	VAR robtarget OpenholeUD_2741 := [[495.65, -37.5, 189.61], [0.203301, 0.677251, 0.701328, -0.090218], [0,0,0,0], [9E9, 9E9, 9E9, 9E9, 9E9, 9E9]];
	VAR robtarget OpenholeUD_2742 := [[499.58, -37.5, 190.31], [0.21303, 0.674254, 0.699718, -0.101956], [0,0,0,0], [9E9, 9E9, 9E9, 9E9, 9E9, 9E9]];
	VAR robtarget OpenholeUD_2743 := [[503.52, -37.5, 191.01], [0.222381, 0.671228, 0.697958, -0.113376], [0,0,0,0], [9E9, 9E9, 9E9, 9E9, 9E9, 9E9]];
	VAR robtarget OpenholeUD_2744 := [[509.38, -37.5, 192.05], [0.183051, 0.683002, 0.683002, -0.183051], [0,0,0,0], [9E9, 9E9, 9E9, 9E9, 9E9, 9E9]];
	VAR robtarget OpenholeUD_2745 := [[513.38, -37.5, 192.04], [0.183051, 0.683002, 0.683002, -0.183051], [0,0,0,0], [9E9, 9E9, 9E9, 9E9, 9E9, 9E9]];
	VAR robtarget OpenholeUD_2746 := [[517.38, -37.5, 192.02], [0.183051, 0.683002, 0.683002, -0.183051], [0,0,0,0], [9E9, 9E9, 9E9, 9E9, 9E9, 9E9]];
	VAR robtarget OpenholeUD_2747 := [[521.38, -37.5, 192.01], [0.183051, 0.683002, 0.683002, -0.183051], [0,0,0,0], [9E9, 9E9, 9E9, 9E9, 9E9, 9E9]];
	VAR robtarget OpenholeUD_2748 := [[525.38, -37.5, 192], [0.183051, 0.683002, 0.683002, -0.183051], [0,0,0,0], [9E9, 9E9, 9E9, 9E9, 9E9, 9E9]];
	VAR robtarget OpenholeUD_2749 := [[529.38, -37.5, 191.99], [0.183051, 0.683002, 0.683002, -0.183051], [0,0,0,0], [9E9, 9E9, 9E9, 9E9, 9E9, 9E9]];
	VAR robtarget OpenholeUD_2750 := [[529.38, -37.5, 191.99], [0.183051, 0.683002, 0.683002, -0.183051], [0,0,0,0], [9E9, 9E9, 9E9, 9E9, 9E9, 9E9]];
	VAR robtarget OpenholeUD_2751 := [[529.38, -38.7, 192.68], [0.183051, 0.683002, 0.683002, -0.183051], [0,0,0,0], [9E9, 9E9, 9E9, 9E9, 9E9, 9E9]];
	VAR robtarget OpenholeUD_2752 := [[525.38, -38.7, 192.69], [0.183051, 0.683002, 0.683002, -0.183051], [0,0,0,0], [9E9, 9E9, 9E9, 9E9, 9E9, 9E9]];
	VAR robtarget OpenholeUD_2753 := [[521.38, -38.7, 192.71], [0.183051, 0.683002, 0.683002, -0.183051], [0,0,0,0], [9E9, 9E9, 9E9, 9E9, 9E9, 9E9]];
	VAR robtarget OpenholeUD_2754 := [[517.38, -38.7, 192.72], [0.183051, 0.683002, 0.683002, -0.183051], [0,0,0,0], [9E9, 9E9, 9E9, 9E9, 9E9, 9E9]];
	VAR robtarget OpenholeUD_2755 := [[513.38, -38.7, 192.73], [0.183051, 0.683002, 0.683002, -0.183051], [0,0,0,0], [9E9, 9E9, 9E9, 9E9, 9E9, 9E9]];
	VAR robtarget OpenholeUD_2756 := [[509.38, -38.7, 192.74], [0.183051, 0.683002, 0.683002, -0.183051], [0,0,0,0], [9E9, 9E9, 9E9, 9E9, 9E9, 9E9]];
	VAR robtarget OpenholeUD_2757 := [[505.45, -38.7, 192], [0.230133, 0.66861, 0.697627, -0.1154], [0,0,0,0], [9E9, 9E9, 9E9, 9E9, 9E9, 9E9]];
	VAR robtarget OpenholeUD_2758 := [[501.52, -38.7, 191.26], [0.221049, 0.671668, 0.699402, -0.104103], [0,0,0,0], [9E9, 9E9, 9E9, 9E9, 9E9, 9E9]];
	VAR robtarget OpenholeUD_2759 := [[497.59, -38.7, 190.51], [0.211589, 0.674707, 0.701032, -0.092485], [0,0,0,0], [9E9, 9E9, 9E9, 9E9, 9E9, 9E9]];
	VAR robtarget OpenholeUD_2760 := [[493.66, -38.7, 189.77], [0.20175, 0.677714, 0.702503, -0.080562], [0,0,0,0], [9E9, 9E9, 9E9, 9E9, 9E9, 9E9]];
	VAR robtarget OpenholeUD_2761 := [[489.73, -38.7, 189.02], [0.191532, 0.680673, 0.703796, -0.06835], [0,0,0,0], [9E9, 9E9, 9E9, 9E9, 9E9, 9E9]];
	VAR robtarget OpenholeUD_2762 := [[485.8, -38.7, 188.28], [0.180935, 0.683566, 0.704896, -0.055873], [0,0,0,0], [9E9, 9E9, 9E9, 9E9, 9E9, 9E9]];
	VAR robtarget OpenholeUD_2763 := [[481.87, -38.7, 187.54], [0.169961, 0.686377, 0.705788, -0.043162], [0,0,0,0], [9E9, 9E9, 9E9, 9E9, 9E9, 9E9]];
	VAR robtarget OpenholeUD_2764 := [[477.94, -38.7, 186.79], [0.158629, 0.689084, 0.70646, -0.030235], [0,0,0,0], [9E9, 9E9, 9E9, 9E9, 9E9, 9E9]];
	VAR robtarget OpenholeUD_2765 := [[474.01, -38.7, 186.05], [0.146953, 0.691668, 0.706899, -0.017125], [0,0,0,0], [9E9, 9E9, 9E9, 9E9, 9E9, 9E9]];
	VAR robtarget OpenholeUD_2766 := [[470.08, -38.7, 185.31], [0.134953, 0.694109, 0.707096, -0.003866], [0,0,0,0], [9E9, 9E9, 9E9, 9E9, 9E9, 9E9]];
	VAR robtarget OpenholeUD_2767 := [[466.15, -38.7, 184.56], [0.122651, 0.696388, 0.707043, 0.009503], [0,0,0,0], [9E9, 9E9, 9E9, 9E9, 9E9, 9E9]];
	VAR robtarget OpenholeUD_2768 := [[462.22, -38.7, 183.82], [0.110074, 0.698487, 0.706735, 0.02294], [0,0,0,0], [9E9, 9E9, 9E9, 9E9, 9E9, 9E9]];
	VAR robtarget OpenholeUD_2769 := [[458.29, -38.7, 183.07], [0.097255, 0.700387, 0.706169, 0.036403], [0,0,0,0], [9E9, 9E9, 9E9, 9E9, 9E9, 9E9]];
	VAR robtarget OpenholeUD_2770 := [[454.36, -38.7, 182.33], [0.084227, 0.702073, 0.705348, 0.049848], [0,0,0,0], [9E9, 9E9, 9E9, 9E9, 9E9, 9E9]];
	VAR robtarget OpenholeUD_2771 := [[450.43, -38.7, 181.59], [0.071029, 0.70353, 0.704274, 0.063232], [0,0,0,0], [9E9, 9E9, 9E9, 9E9, 9E9, 9E9]];
	VAR robtarget OpenholeUD_2772 := [[446.5, -38.7, 180.84], [0.05769, 0.70475, 0.702956, 0.0765], [0,0,0,0], [9E9, 9E9, 9E9, 9E9, 9E9, 9E9]];
	VAR robtarget OpenholeUD_2773 := [[442.57, -38.7, 180.1], [0.044257, 0.70572, 0.701405, 0.089614], [0,0,0,0], [9E9, 9E9, 9E9, 9E9, 9E9, 9E9]];
	VAR robtarget OpenholeUD_2774 := [[438.64, -38.7, 179.35], [0.030777, 0.706437, 0.699632, 0.102541], [0,0,0,0], [9E9, 9E9, 9E9, 9E9, 9E9, 9E9]];
	VAR robtarget OpenholeUD_2775 := [[434.71, -38.7, 178.61], [0.017296, 0.706895, 0.697653, 0.115242], [0,0,0,0], [9E9, 9E9, 9E9, 9E9, 9E9, 9E9]];
	VAR robtarget OpenholeUD_2776 := [[430.78, -38.7, 177.87], [0.003855, 0.707096, 0.695483, 0.127685], [0,0,0,0], [9E9, 9E9, 9E9, 9E9, 9E9, 9E9]];
	VAR robtarget OpenholeUD_2777 := [[426.85, -38.7, 177.12], [-0.009501, 0.707043, 0.693141, 0.139841], [0,0,0,0], [9E9, 9E9, 9E9, 9E9, 9E9, 9E9]];
	VAR robtarget OpenholeUD_2778 := [[422.92, -38.7, 176.38], [-0.022733, 0.706741, 0.690646, 0.151685], [0,0,0,0], [9E9, 9E9, 9E9, 9E9, 9E9, 9E9]];
	VAR robtarget OpenholeUD_2779 := [[418.99, -38.7, 175.64], [-0.035803, 0.7062, 0.688017, 0.163195], [0,0,0,0], [9E9, 9E9, 9E9, 9E9, 9E9, 9E9]];
	VAR robtarget OpenholeUD_2780 := [[415.06, -38.7, 174.89], [-0.048676, 0.705429, 0.685274, 0.174356], [0,0,0,0], [9E9, 9E9, 9E9, 9E9, 9E9, 9E9]];
	VAR robtarget OpenholeUD_2781 := [[411.13, -38.7, 174.15], [-0.061321, 0.704443, 0.682435, 0.185154], [0,0,0,0], [9E9, 9E9, 9E9, 9E9, 9E9, 9E9]];
	VAR robtarget OpenholeUD_2782 := [[407.2, -38.7, 173.4], [-0.073711, 0.703254, 0.67952, 0.195582], [0,0,0,0], [9E9, 9E9, 9E9, 9E9, 9E9, 9E9]];
	VAR robtarget OpenholeUD_2783 := [[403.27, -38.7, 172.66], [-0.085821, 0.701879, 0.676546, 0.205634], [0,0,0,0], [9E9, 9E9, 9E9, 9E9, 9E9, 9E9]];
	VAR robtarget OpenholeUD_2784 := [[399.34, -38.7, 171.92], [-0.097632, 0.700334, 0.67353, 0.215308], [0,0,0,0], [9E9, 9E9, 9E9, 9E9, 9E9, 9E9]];
	VAR robtarget OpenholeUD_2785 := [[395.41, -38.7, 171.17], [-0.109129, 0.698635, 0.670487, 0.224606], [0,0,0,0], [9E9, 9E9, 9E9, 9E9, 9E9, 9E9]];
	VAR robtarget OpenholeUD_2786 := [[389.31, -38.7, 170.02], [-0.126309, 0.695734, 0.665746, 0.238291], [0,0,0,0], [9E9, 9E9, 9E9, 9E9, 9E9, 9E9]];
	VAR robtarget OpenholeUD_2787 := [[385.31, -38.7, 170.03], [-0.183051, 0.683002, 0.683002, 0.183051], [0,0,0,0], [9E9, 9E9, 9E9, 9E9, 9E9, 9E9]];
	VAR robtarget OpenholeUD_2788 := [[381.31, -38.7, 170.05], [-0.183051, 0.683002, 0.683002, 0.183051], [0,0,0,0], [9E9, 9E9, 9E9, 9E9, 9E9, 9E9]];
	VAR robtarget OpenholeUD_2789 := [[377.31, -38.7, 170.06], [-0.183051, 0.683002, 0.683002, 0.183051], [0,0,0,0], [9E9, 9E9, 9E9, 9E9, 9E9, 9E9]];
	VAR robtarget OpenholeUD_2790 := [[373.31, -38.7, 170.07], [-0.183051, 0.683002, 0.683002, 0.183051], [0,0,0,0], [9E9, 9E9, 9E9, 9E9, 9E9, 9E9]];
	VAR robtarget OpenholeUD_2791 := [[369.31, -38.7, 170.08], [-0.183051, 0.683002, 0.683002, 0.183051], [0,0,0,0], [9E9, 9E9, 9E9, 9E9, 9E9, 9E9]];
	VAR robtarget OpenholeUD_2792 := [[369.31, -38.7, 170.08], [-0.183051, 0.683002, 0.683002, 0.183051], [0,0,0,0], [9E9, 9E9, 9E9, 9E9, 9E9, 9E9]];
	VAR robtarget OpenholeUD_2793 := [[369.31, -38.7, 170.2], [-0.183051, 0.683002, 0.683002, 0.183051], [0,0,0,0], [9E9, 9E9, 9E9, 9E9, 9E9, 9E9]];
	VAR robtarget OpenholeUD_2794 := [[373.31, -38.7, 170.19], [-0.183051, 0.683002, 0.683002, 0.183051], [0,0,0,0], [9E9, 9E9, 9E9, 9E9, 9E9, 9E9]];
	VAR robtarget OpenholeUD_2795 := [[377.31, -38.7, 170.18], [-0.183051, 0.683002, 0.683002, 0.183051], [0,0,0,0], [9E9, 9E9, 9E9, 9E9, 9E9, 9E9]];
	VAR robtarget OpenholeUD_2796 := [[381.31, -38.7, 170.17], [-0.183051, 0.683002, 0.683002, 0.183051], [0,0,0,0], [9E9, 9E9, 9E9, 9E9, 9E9, 9E9]];
	VAR robtarget OpenholeUD_2797 := [[385.31, -38.7, 170.15], [-0.183051, 0.683002, 0.683002, 0.183051], [0,0,0,0], [9E9, 9E9, 9E9, 9E9, 9E9, 9E9]];
	VAR robtarget OpenholeUD_2798 := [[389.31, -38.7, 170.14], [-0.126405, 0.695717, 0.665808, 0.238118], [0,0,0,0], [9E9, 9E9, 9E9, 9E9, 9E9, 9E9]];
	VAR robtarget OpenholeUD_2799 := [[393.24, -38.7, 170.88], [-0.115413, 0.697624, 0.668864, 0.229394], [0,0,0,0], [9E9, 9E9, 9E9, 9E9, 9E9, 9E9]];
	VAR robtarget OpenholeUD_2800 := [[397.17, -38.7, 171.63], [-0.104088, 0.699404, 0.671913, 0.220302], [0,0,0,0], [9E9, 9E9, 9E9, 9E9, 9E9, 9E9]];
	VAR robtarget OpenholeUD_2801 := [[401.1, -38.7, 172.37], [-0.092441, 0.701038, 0.674943, 0.210836], [0,0,0,0], [9E9, 9E9, 9E9, 9E9, 9E9, 9E9]];
	VAR robtarget OpenholeUD_2802 := [[405.03, -38.7, 173.12], [-0.080484, 0.702511, 0.677939, 0.200994], [0,0,0,0], [9E9, 9E9, 9E9, 9E9, 9E9, 9E9]];
	VAR robtarget OpenholeUD_2803 := [[408.96, -38.7, 173.86], [-0.068237, 0.703807, 0.680885, 0.190776], [0,0,0,0], [9E9, 9E9, 9E9, 9E9, 9E9, 9E9]];
	VAR robtarget OpenholeUD_2804 := [[412.89, -38.7, 174.6], [-0.055719, 0.704908, 0.683764, 0.180185], [0,0,0,0], [9E9, 9E9, 9E9, 9E9, 9E9, 9E9]];
	VAR robtarget OpenholeUD_2805 := [[416.82, -38.7, 175.35], [-0.042956, 0.705801, 0.686558, 0.169228], [0,0,0,0], [9E9, 9E9, 9E9, 9E9, 9E9, 9E9]];
	VAR robtarget OpenholeUD_2806 := [[420.75, -38.7, 176.09], [-0.029979, 0.706471, 0.689248, 0.157914], [0,0,0,0], [9E9, 9E9, 9E9, 9E9, 9E9, 9E9]];
	VAR robtarget OpenholeUD_2807 := [[424.68, -38.7, 176.83], [-0.016818, 0.706907, 0.691815, 0.146259], [0,0,0,0], [9E9, 9E9, 9E9, 9E9, 9E9, 9E9]];
	VAR robtarget OpenholeUD_2808 := [[428.61, -38.7, 177.58], [-0.003512, 0.707098, 0.69424, 0.13428], [0,0,0,0], [9E9, 9E9, 9E9, 9E9, 9E9, 9E9]];
	VAR robtarget OpenholeUD_2809 := [[432.54, -38.7, 178.32], [0.009901, 0.707037, 0.696502, 0.122002], [0,0,0,0], [9E9, 9E9, 9E9, 9E9, 9E9, 9E9]];
	VAR robtarget OpenholeUD_2810 := [[436.47, -38.7, 179.07], [0.02338, 0.70672, 0.698585, 0.109449], [0,0,0,0], [9E9, 9E9, 9E9, 9E9, 9E9, 9E9]];
	VAR robtarget OpenholeUD_2811 := [[440.4, -38.7, 179.81], [0.036881, 0.706144, 0.70047, 0.096654], [0,0,0,0], [9E9, 9E9, 9E9, 9E9, 9E9, 9E9]];
	VAR robtarget OpenholeUD_2812 := [[444.33, -38.7, 180.55], [0.050359, 0.705311, 0.702141, 0.083651], [0,0,0,0], [9E9, 9E9, 9E9, 9E9, 9E9, 9E9]];
	VAR robtarget OpenholeUD_2813 := [[448.26, -38.7, 181.3], [0.063771, 0.704225, 0.703586, 0.070478], [0,0,0,0], [9E9, 9E9, 9E9, 9E9, 9E9, 9E9]];
	VAR robtarget OpenholeUD_2814 := [[452.19, -38.7, 182.04], [0.077052, 0.702896, 0.704793, 0.057153], [0,0,0,0], [9E9, 9E9, 9E9, 9E9, 9E9, 9E9]];
	VAR robtarget OpenholeUD_2815 := [[456.12, -38.7, 182.78], [0.090178, 0.701333, 0.705753, 0.043736], [0,0,0,0], [9E9, 9E9, 9E9, 9E9, 9E9, 9E9]];
	VAR robtarget OpenholeUD_2816 := [[460.06, -38.7, 183.53], [0.103115, 0.699548, 0.706458, 0.030277], [0,0,0,0], [9E9, 9E9, 9E9, 9E9, 9E9, 9E9]];
	VAR robtarget OpenholeUD_2817 := [[463.99, -38.7, 184.27], [0.115828, 0.697556, 0.706907, 0.01682], [0,0,0,0], [9E9, 9E9, 9E9, 9E9, 9E9, 9E9]];
	VAR robtarget OpenholeUD_2818 := [[467.92, -38.7, 185.02], [0.128284, 0.695373, 0.707099, 0.003409], [0,0,0,0], [9E9, 9E9, 9E9, 9E9, 9E9, 9E9]];
	VAR robtarget OpenholeUD_2819 := [[471.85, -38.7, 185.76], [0.140451, 0.693018, 0.707037, -0.009914], [0,0,0,0], [9E9, 9E9, 9E9, 9E9, 9E9, 9E9]];
	VAR robtarget OpenholeUD_2820 := [[475.78, -38.7, 186.5], [0.152307, 0.690509, 0.706729, -0.02311], [0,0,0,0], [9E9, 9E9, 9E9, 9E9, 9E9, 9E9]];
	VAR robtarget OpenholeUD_2821 := [[479.71, -38.7, 187.25], [0.163828, 0.687867, 0.706183, -0.036142], [0,0,0,0], [9E9, 9E9, 9E9, 9E9, 9E9, 9E9]];
	VAR robtarget OpenholeUD_2822 := [[483.64, -38.7, 187.99], [0.174999, 0.68511, 0.705409, -0.048974], [0,0,0,0], [9E9, 9E9, 9E9, 9E9, 9E9, 9E9]];
	VAR robtarget OpenholeUD_2823 := [[487.57, -38.7, 188.73], [0.185806, 0.682258, 0.704421, -0.061577], [0,0,0,0], [9E9, 9E9, 9E9, 9E9, 9E9, 9E9]];
	VAR robtarget OpenholeUD_2824 := [[491.5, -38.7, 189.48], [0.196242, 0.67933, 0.703232, -0.073924], [0,0,0,0], [9E9, 9E9, 9E9, 9E9, 9E9, 9E9]];
	VAR robtarget OpenholeUD_2825 := [[495.43, -38.7, 190.22], [0.2063, 0.676343, 0.701859, -0.085991], [0,0,0,0], [9E9, 9E9, 9E9, 9E9, 9E9, 9E9]];
	VAR robtarget OpenholeUD_2826 := [[499.36, -38.7, 190.97], [0.21598, 0.673315, 0.700316, -0.09776], [0,0,0,0], [9E9, 9E9, 9E9, 9E9, 9E9, 9E9]];
	VAR robtarget OpenholeUD_2827 := [[503.29, -38.7, 191.71], [0.225282, 0.67026, 0.698621, -0.109216], [0,0,0,0], [9E9, 9E9, 9E9, 9E9, 9E9, 9E9]];
	VAR robtarget OpenholeUD_2828 := [[509.38, -38.7, 192.86], [0.183051, 0.683002, 0.683002, -0.183051], [0,0,0,0], [9E9, 9E9, 9E9, 9E9, 9E9, 9E9]];
	VAR robtarget OpenholeUD_2829 := [[513.38, -38.7, 192.85], [0.183051, 0.683002, 0.683002, -0.183051], [0,0,0,0], [9E9, 9E9, 9E9, 9E9, 9E9, 9E9]];
	VAR robtarget OpenholeUD_2830 := [[517.38, -38.7, 192.84], [0.183051, 0.683002, 0.683002, -0.183051], [0,0,0,0], [9E9, 9E9, 9E9, 9E9, 9E9, 9E9]];
	VAR robtarget OpenholeUD_2831 := [[521.38, -38.7, 192.83], [0.183051, 0.683002, 0.683002, -0.183051], [0,0,0,0], [9E9, 9E9, 9E9, 9E9, 9E9, 9E9]];
	VAR robtarget OpenholeUD_2832 := [[525.38, -38.7, 192.81], [0.183051, 0.683002, 0.683002, -0.183051], [0,0,0,0], [9E9, 9E9, 9E9, 9E9, 9E9, 9E9]];
	VAR robtarget OpenholeUD_2833 := [[529.38, -38.7, 192.8], [0.183051, 0.683002, 0.683002, -0.183051], [0,0,0,0], [9E9, 9E9, 9E9, 9E9, 9E9, 9E9]];
	VAR robtarget OpenholeUD_2834 := [[529.38, -38.7, 192.8], [0.183051, 0.683002, 0.683002, -0.183051], [0,0,0,0], [9E9, 9E9, 9E9, 9E9, 9E9, 9E9]];
	VAR robtarget OpenholeUD_2835 := [[529.38, -37.5, 192.11], [0.183051, 0.683002, 0.683002, -0.183051], [0,0,0,0], [9E9, 9E9, 9E9, 9E9, 9E9, 9E9]];
	VAR robtarget OpenholeUD_2836 := [[525.38, -37.5, 192.12], [0.183051, 0.683002, 0.683002, -0.183051], [0,0,0,0], [9E9, 9E9, 9E9, 9E9, 9E9, 9E9]];
	VAR robtarget OpenholeUD_2837 := [[521.38, -37.5, 192.13], [0.183051, 0.683002, 0.683002, -0.183051], [0,0,0,0], [9E9, 9E9, 9E9, 9E9, 9E9, 9E9]];
	VAR robtarget OpenholeUD_2838 := [[517.38, -37.5, 192.14], [0.183051, 0.683002, 0.683002, -0.183051], [0,0,0,0], [9E9, 9E9, 9E9, 9E9, 9E9, 9E9]];
	VAR robtarget OpenholeUD_2839 := [[513.38, -37.5, 192.16], [0.183051, 0.683002, 0.683002, -0.183051], [0,0,0,0], [9E9, 9E9, 9E9, 9E9, 9E9, 9E9]];
	VAR robtarget OpenholeUD_2840 := [[509.38, -37.5, 192.17], [0.183051, 0.683002, 0.683002, -0.183051], [0,0,0,0], [9E9, 9E9, 9E9, 9E9, 9E9, 9E9]];
	VAR robtarget OpenholeUD_2841 := [[505.44, -37.5, 191.47], [0.226975, 0.669688, 0.697068, -0.118728], [0,0,0,0], [9E9, 9E9, 9E9, 9E9, 9E9, 9E9]];
	VAR robtarget OpenholeUD_2842 := [[501.5, -37.5, 190.77], [0.217806, 0.672726, 0.698892, -0.107473], [0,0,0,0], [9E9, 9E9, 9E9, 9E9, 9E9, 9E9]];
	VAR robtarget OpenholeUD_2843 := [[497.57, -37.5, 190.07], [0.20826, 0.675742, 0.700574, -0.095895], [0,0,0,0], [9E9, 9E9, 9E9, 9E9, 9E9, 9E9]];
	VAR robtarget OpenholeUD_2844 := [[493.63, -37.5, 189.37], [0.198335, 0.678722, 0.702099, -0.084008], [0,0,0,0], [9E9, 9E9, 9E9, 9E9, 9E9, 9E9]];
	VAR robtarget OpenholeUD_2845 := [[489.69, -37.5, 188.67], [0.18803, 0.681649, 0.703449, -0.07183], [0,0,0,0], [9E9, 9E9, 9E9, 9E9, 9E9, 9E9]];
	VAR robtarget OpenholeUD_2846 := [[485.75, -37.5, 187.97], [0.177348, 0.684505, 0.704609, -0.05938], [0,0,0,0], [9E9, 9E9, 9E9, 9E9, 9E9, 9E9]];
	VAR robtarget OpenholeUD_2847 := [[481.81, -37.5, 187.27], [0.166298, 0.687274, 0.705564, -0.046684], [0,0,0,0], [9E9, 9E9, 9E9, 9E9, 9E9, 9E9]];
	VAR robtarget OpenholeUD_2848 := [[477.87, -37.5, 186.57], [0.154888, 0.689935, 0.7063, -0.03377], [0,0,0,0], [9E9, 9E9, 9E9, 9E9, 9E9, 9E9]];
	VAR robtarget OpenholeUD_2849 := [[473.94, -37.5, 185.87], [0.143135, 0.692468, 0.706805, -0.020671], [0,0,0,0], [9E9, 9E9, 9E9, 9E9, 9E9, 9E9]];
	VAR robtarget OpenholeUD_2850 := [[470, -37.5, 185.17], [0.131057, 0.694855, 0.707068, -0.007421], [0,0,0,0], [9E9, 9E9, 9E9, 9E9, 9E9, 9E9]];
	VAR robtarget OpenholeUD_2851 := [[466.06, -37.5, 184.47], [0.118677, 0.697077, 0.707082, 0.005939], [0,0,0,0], [9E9, 9E9, 9E9, 9E9, 9E9, 9E9]];
	VAR robtarget OpenholeUD_2852 := [[462.12, -37.5, 183.77], [0.106025, 0.699113, 0.706841, 0.01937], [0,0,0,0], [9E9, 9E9, 9E9, 9E9, 9E9, 9E9]];
	VAR robtarget OpenholeUD_2853 := [[458.18, -37.5, 183.07], [0.093131, 0.700947, 0.706344, 0.03283], [0,0,0,0], [9E9, 9E9, 9E9, 9E9, 9E9, 9E9]];
	VAR robtarget OpenholeUD_2854 := [[454.24, -37.5, 182.37], [0.08003, 0.702563, 0.705591, 0.046273], [0,0,0,0], [9E9, 9E9, 9E9, 9E9, 9E9, 9E9]];
	VAR robtarget OpenholeUD_2855 := [[450.31, -37.5, 181.67], [0.066762, 0.703948, 0.704586, 0.059657], [0,0,0,0], [9E9, 9E9, 9E9, 9E9, 9E9, 9E9]];
	VAR robtarget OpenholeUD_2856 := [[446.37, -37.5, 180.97], [0.053369, 0.70509, 0.703335, 0.072939], [0,0,0,0], [9E9, 9E9, 9E9, 9E9, 9E9, 9E9]];
	VAR robtarget OpenholeUD_2857 := [[442.43, -37.5, 180.27], [0.039892, 0.705981, 0.701848, 0.086077], [0,0,0,0], [9E9, 9E9, 9E9, 9E9, 9E9, 9E9]];
	VAR robtarget OpenholeUD_2858 := [[438.49, -37.5, 179.57], [0.026377, 0.706615, 0.700138, 0.099031], [0,0,0,0], [9E9, 9E9, 9E9, 9E9, 9E9, 9E9]];
	VAR robtarget OpenholeUD_2859 := [[434.55, -37.5, 178.87], [0.012867, 0.70699, 0.698218, 0.111765], [0,0,0,0], [9E9, 9E9, 9E9, 9E9, 9E9, 9E9]];
	VAR robtarget OpenholeUD_2860 := [[430.61, -37.5, 178.17], [-0.000592, 0.707107, 0.696106, 0.124246], [0,0,0,0], [9E9, 9E9, 9E9, 9E9, 9E9, 9E9]];
	VAR robtarget OpenholeUD_2861 := [[426.68, -37.5, 177.47], [-0.013959, 0.706969, 0.693818, 0.136443], [0,0,0,0], [9E9, 9E9, 9E9, 9E9, 9E9, 9E9]];
	VAR robtarget OpenholeUD_2862 := [[422.74, -37.5, 176.77], [-0.027193, 0.706584, 0.691374, 0.148332], [0,0,0,0], [9E9, 9E9, 9E9, 9E9, 9E9, 9E9]];
	VAR robtarget OpenholeUD_2863 := [[418.8, -37.5, 176.07], [-0.040257, 0.70596, 0.688792, 0.159891], [0,0,0,0], [9E9, 9E9, 9E9, 9E9, 9E9, 9E9]];
	VAR robtarget OpenholeUD_2864 := [[414.86, -37.5, 175.37], [-0.053115, 0.705109, 0.686093, 0.171103], [0,0,0,0], [9E9, 9E9, 9E9, 9E9, 9E9, 9E9]];
	VAR robtarget OpenholeUD_2865 := [[410.92, -37.5, 174.67], [-0.065738, 0.704044, 0.683295, 0.181955], [0,0,0,0], [9E9, 9E9, 9E9, 9E9, 9E9, 9E9]];
	VAR robtarget OpenholeUD_2866 := [[406.98, -37.5, 173.97], [-0.078098, 0.702781, 0.680417, 0.192438], [0,0,0,0], [9E9, 9E9, 9E9, 9E9, 9E9, 9E9]];
	VAR robtarget OpenholeUD_2867 := [[403.05, -37.5, 173.27], [-0.090172, 0.701334, 0.677477, 0.202547], [0,0,0,0], [9E9, 9E9, 9E9, 9E9, 9E9, 9E9]];
	VAR robtarget OpenholeUD_2868 := [[399.11, -37.5, 172.57], [-0.101941, 0.69972, 0.67449, 0.21228], [0,0,0,0], [9E9, 9E9, 9E9, 9E9, 9E9, 9E9]];
	VAR robtarget OpenholeUD_2869 := [[395.17, -37.5, 171.87], [-0.113391, 0.697956, 0.671473, 0.221638], [0,0,0,0], [9E9, 9E9, 9E9, 9E9, 9E9, 9E9]];
	VAR robtarget OpenholeUD_2870 := [[389.31, -37.5, 170.83], [-0.129802, 0.695091, 0.666961, 0.234869], [0,0,0,0], [9E9, 9E9, 9E9, 9E9, 9E9, 9E9]];
	VAR robtarget OpenholeUD_2871 := [[385.31, -37.5, 170.85], [-0.183051, 0.683002, 0.683002, 0.183051], [0,0,0,0], [9E9, 9E9, 9E9, 9E9, 9E9, 9E9]];
	VAR robtarget OpenholeUD_2872 := [[381.31, -37.5, 170.86], [-0.183051, 0.683002, 0.683002, 0.183051], [0,0,0,0], [9E9, 9E9, 9E9, 9E9, 9E9, 9E9]];
	VAR robtarget OpenholeUD_2873 := [[377.31, -37.5, 170.87], [-0.183051, 0.683002, 0.683002, 0.183051], [0,0,0,0], [9E9, 9E9, 9E9, 9E9, 9E9, 9E9]];
	VAR robtarget OpenholeUD_2874 := [[373.31, -37.5, 170.88], [-0.183051, 0.683002, 0.683002, 0.183051], [0,0,0,0], [9E9, 9E9, 9E9, 9E9, 9E9, 9E9]];
	VAR robtarget OpenholeUD_2875 := [[369.31, -37.5, 170.9], [-0.183051, 0.683002, 0.683002, 0.183051], [0,0,0,0], [9E9, 9E9, 9E9, 9E9, 9E9, 9E9]];
	VAR robtarget OpenholeUD_2876 := [[369.31, -37.5, 170.9], [-0.183051, 0.683002, 0.683002, 0.183051], [0,0,0,0], [9E9, 9E9, 9E9, 9E9, 9E9, 9E9]];
	VAR robtarget OpenholeUD_2877 := [[369.32, -36.3, 171.59], [-0.183051, 0.683002, 0.683002, 0.183051], [0,0,0,0], [9E9, 9E9, 9E9, 9E9, 9E9, 9E9]];
	VAR robtarget OpenholeUD_2878 := [[373.32, -36.3, 171.58], [-0.183051, 0.683002, 0.683002, 0.183051], [0,0,0,0], [9E9, 9E9, 9E9, 9E9, 9E9, 9E9]];
	VAR robtarget OpenholeUD_2879 := [[377.32, -36.3, 171.56], [-0.183051, 0.683002, 0.683002, 0.183051], [0,0,0,0], [9E9, 9E9, 9E9, 9E9, 9E9, 9E9]];
	VAR robtarget OpenholeUD_2880 := [[381.32, -36.3, 171.55], [-0.183051, 0.683002, 0.683002, 0.183051], [0,0,0,0], [9E9, 9E9, 9E9, 9E9, 9E9, 9E9]];
	VAR robtarget OpenholeUD_2881 := [[385.32, -36.3, 171.54], [-0.183051, 0.683002, 0.683002, 0.183051], [0,0,0,0], [9E9, 9E9, 9E9, 9E9, 9E9, 9E9]];
	VAR robtarget OpenholeUD_2882 := [[389.32, -36.3, 171.53], [-0.133206, 0.694447, 0.668101, 0.231606], [0,0,0,0], [9E9, 9E9, 9E9, 9E9, 9E9, 9E9]];
	VAR robtarget OpenholeUD_2883 := [[393.26, -36.3, 172.18], [-0.122294, 0.696451, 0.671117, 0.222715], [0,0,0,0], [9E9, 9E9, 9E9, 9E9, 9E9, 9E9]];
	VAR robtarget OpenholeUD_2884 := [[397.21, -36.3, 172.84], [-0.111044, 0.698333, 0.674119, 0.213456], [0,0,0,0], [9E9, 9E9, 9E9, 9E9, 9E9, 9E9]];
	VAR robtarget OpenholeUD_2885 := [[401.15, -36.3, 173.49], [-0.099464, 0.700076, 0.677094, 0.203822], [0,0,0,0], [9E9, 9E9, 9E9, 9E9, 9E9, 9E9]];
	VAR robtarget OpenholeUD_2886 := [[405.1, -36.3, 174.15], [-0.087567, 0.701664, 0.680027, 0.193813], [0,0,0,0], [9E9, 9E9, 9E9, 9E9, 9E9, 9E9]];
	VAR robtarget OpenholeUD_2887 := [[409.04, -36.3, 174.8], [-0.075371, 0.703078, 0.682901, 0.183428], [0,0,0,0], [9E9, 9E9, 9E9, 9E9, 9E9, 9E9]];
	VAR robtarget OpenholeUD_2888 := [[412.99, -36.3, 175.46], [-0.062895, 0.704304, 0.685699, 0.172674], [0,0,0,0], [9E9, 9E9, 9E9, 9E9, 9E9, 9E9]];
	VAR robtarget OpenholeUD_2889 := [[416.94, -36.3, 176.12], [-0.050166, 0.705325, 0.688404, 0.161556], [0,0,0,0], [9E9, 9E9, 9E9, 9E9, 9E9, 9E9]];
	VAR robtarget OpenholeUD_2890 := [[420.88, -36.3, 176.77], [-0.03721, 0.706127, 0.690995, 0.150088], [0,0,0,0], [9E9, 9E9, 9E9, 9E9, 9E9, 9E9]];
	VAR robtarget OpenholeUD_2891 := [[424.83, -36.3, 177.43], [-0.024062, 0.706697, 0.693453, 0.138284], [0,0,0,0], [9E9, 9E9, 9E9, 9E9, 9E9, 9E9]];
	VAR robtarget OpenholeUD_2892 := [[428.77, -36.3, 178.08], [-0.010756, 0.707025, 0.69576, 0.126164], [0,0,0,0], [9E9, 9E9, 9E9, 9E9, 9E9, 9E9]];
	VAR robtarget OpenholeUD_2893 := [[432.72, -36.3, 178.74], [0.002667, 0.707102, 0.697897, 0.113753], [0,0,0,0], [9E9, 9E9, 9E9, 9E9, 9E9, 9E9]];
	VAR robtarget OpenholeUD_2894 := [[436.67, -36.3, 179.39], [0.016167, 0.706922, 0.699845, 0.101079], [0,0,0,0], [9E9, 9E9, 9E9, 9E9, 9E9, 9E9]];
	VAR robtarget OpenholeUD_2895 := [[440.61, -36.3, 180.05], [0.029701, 0.706483, 0.701588, 0.088173], [0,0,0,0], [9E9, 9E9, 9E9, 9E9, 9E9, 9E9]];
	VAR robtarget OpenholeUD_2896 := [[444.56, -36.3, 180.71], [0.043222, 0.705785, 0.70311, 0.075072], [0,0,0,0], [9E9, 9E9, 9E9, 9E9, 9E9, 9E9]];
	VAR robtarget OpenholeUD_2897 := [[448.5, -36.3, 181.36], [0.056688, 0.704831, 0.7044, 0.061815], [0,0,0,0], [9E9, 9E9, 9E9, 9E9, 9E9, 9E9]];
	VAR robtarget OpenholeUD_2898 := [[452.45, -36.3, 182.02], [0.070054, 0.703628, 0.705446, 0.048442], [0,0,0,0], [9E9, 9E9, 9E9, 9E9, 9E9, 9E9]];
	VAR robtarget OpenholeUD_2899 := [[456.4, -36.3, 182.67], [0.083277, 0.702186, 0.70624, 0.034996], [0,0,0,0], [9E9, 9E9, 9E9, 9E9, 9E9, 9E9]];
	VAR robtarget OpenholeUD_2900 := [[460.34, -36.3, 183.33], [0.096317, 0.700516, 0.706779, 0.021521], [0,0,0,0], [9E9, 9E9, 9E9, 9E9, 9E9, 9E9]];
	VAR robtarget OpenholeUD_2901 := [[464.29, -36.3, 183.98], [0.109136, 0.698634, 0.707061, 0.008061], [0,0,0,0], [9E9, 9E9, 9E9, 9E9, 9E9, 9E9]];
	VAR robtarget OpenholeUD_2902 := [[468.23, -36.3, 184.64], [0.1217, 0.696555, 0.707087, -0.005341], [0,0,0,0], [9E9, 9E9, 9E9, 9E9, 9E9, 9E9]];
	VAR robtarget OpenholeUD_2903 := [[472.18, -36.3, 185.3], [0.133979, 0.694298, 0.706861, -0.018643], [0,0,0,0], [9E9, 9E9, 9E9, 9E9, 9E9, 9E9]];
	VAR robtarget OpenholeUD_2904 := [[476.12, -36.3, 185.95], [0.145948, 0.691881, 0.706391, -0.031805], [0,0,0,0], [9E9, 9E9, 9E9, 9E9, 9E9, 9E9]];
	VAR robtarget OpenholeUD_2905 := [[480.07, -36.3, 186.61], [0.157583, 0.689324, 0.705687, -0.044792], [0,0,0,0], [9E9, 9E9, 9E9, 9E9, 9E9, 9E9]];
	VAR robtarget OpenholeUD_2906 := [[484.02, -36.3, 187.26], [0.168868, 0.686647, 0.704759, -0.05757], [0,0,0,0], [9E9, 9E9, 9E9, 9E9, 9E9, 9E9]];
	VAR robtarget OpenholeUD_2907 := [[487.96, -36.3, 187.92], [0.17979, 0.683868, 0.703623, -0.070108], [0,0,0,0], [9E9, 9E9, 9E9, 9E9, 9E9, 9E9]];
	VAR robtarget OpenholeUD_2908 := [[491.91, -36.3, 188.57], [0.19034, 0.681007, 0.702292, -0.08238], [0,0,0,0], [9E9, 9E9, 9E9, 9E9, 9E9, 9E9]];
	VAR robtarget OpenholeUD_2909 := [[495.85, -36.3, 189.23], [0.200512, 0.678082, 0.700782, -0.094365], [0,0,0,0], [9E9, 9E9, 9E9, 9E9, 9E9, 9E9]];
	VAR robtarget OpenholeUD_2910 := [[499.8, -36.3, 189.89], [0.210305, 0.675109, 0.69911, -0.106044], [0,0,0,0], [9E9, 9E9, 9E9, 9E9, 9E9, 9E9]];
	VAR robtarget OpenholeUD_2911 := [[503.75, -36.3, 190.54], [0.219719, 0.672104, 0.697293, -0.117402], [0,0,0,0], [9E9, 9E9, 9E9, 9E9, 9E9, 9E9]];
	VAR robtarget OpenholeUD_2912 := [[509.38, -36.3, 191.48], [0.183051, 0.683002, 0.683002, -0.183051], [0,0,0,0], [9E9, 9E9, 9E9, 9E9, 9E9, 9E9]];
	VAR robtarget OpenholeUD_2913 := [[513.38, -36.3, 191.46], [0.183051, 0.683002, 0.683002, -0.183051], [0,0,0,0], [9E9, 9E9, 9E9, 9E9, 9E9, 9E9]];
	VAR robtarget OpenholeUD_2914 := [[517.38, -36.3, 191.45], [0.183051, 0.683002, 0.683002, -0.183051], [0,0,0,0], [9E9, 9E9, 9E9, 9E9, 9E9, 9E9]];
	VAR robtarget OpenholeUD_2915 := [[521.38, -36.3, 191.44], [0.183051, 0.683002, 0.683002, -0.183051], [0,0,0,0], [9E9, 9E9, 9E9, 9E9, 9E9, 9E9]];
	VAR robtarget OpenholeUD_2916 := [[525.38, -36.3, 191.43], [0.183051, 0.683002, 0.683002, -0.183051], [0,0,0,0], [9E9, 9E9, 9E9, 9E9, 9E9, 9E9]];
	VAR robtarget OpenholeUD_2917 := [[529.38, -36.3, 191.41], [0.183051, 0.683002, 0.683002, -0.183051], [0,0,0,0], [9E9, 9E9, 9E9, 9E9, 9E9, 9E9]];
	VAR robtarget OpenholeUD_2918 := [[529.38, -36.3, 191.41], [0.183051, 0.683002, 0.683002, -0.183051], [0,0,0,0], [9E9, 9E9, 9E9, 9E9, 9E9, 9E9]];
	VAR robtarget OpenholeUD_2919 := [[529.38, -35.1, 190.72], [0.183051, 0.683002, 0.683002, -0.183051], [0,0,0,0], [9E9, 9E9, 9E9, 9E9, 9E9, 9E9]];
	VAR robtarget OpenholeUD_2920 := [[525.38, -35.1, 190.73], [0.183051, 0.683002, 0.683002, -0.183051], [0,0,0,0], [9E9, 9E9, 9E9, 9E9, 9E9, 9E9]];
	VAR robtarget OpenholeUD_2921 := [[521.38, -35.1, 190.75], [0.183051, 0.683002, 0.683002, -0.183051], [0,0,0,0], [9E9, 9E9, 9E9, 9E9, 9E9, 9E9]];
	VAR robtarget OpenholeUD_2922 := [[517.38, -35.1, 190.76], [0.183051, 0.683002, 0.683002, -0.183051], [0,0,0,0], [9E9, 9E9, 9E9, 9E9, 9E9, 9E9]];
	VAR robtarget OpenholeUD_2923 := [[513.38, -35.1, 190.77], [0.183051, 0.683002, 0.683002, -0.183051], [0,0,0,0], [9E9, 9E9, 9E9, 9E9, 9E9, 9E9]];
	VAR robtarget OpenholeUD_2924 := [[509.38, -35.1, 190.78], [0.183051, 0.683002, 0.683002, -0.183051], [0,0,0,0], [9E9, 9E9, 9E9, 9E9, 9E9, 9E9]];
	VAR robtarget OpenholeUD_2925 := [[505.42, -35.1, 190.17], [0.220265, 0.671925, 0.695864, -0.125592], [0,0,0,0], [9E9, 9E9, 9E9, 9E9, 9E9, 9E9]];
	VAR robtarget OpenholeUD_2926 := [[501.47, -35.1, 189.56], [0.210928, 0.674914, 0.697789, -0.114414], [0,0,0,0], [9E9, 9E9, 9E9, 9E9, 9E9, 9E9]];
	VAR robtarget OpenholeUD_2927 := [[497.52, -35.1, 188.95], [0.201214, 0.677874, 0.699578, -0.102908], [0,0,0,0], [9E9, 9E9, 9E9, 9E9, 9E9, 9E9]];
	VAR robtarget OpenholeUD_2928 := [[493.56, -35.1, 188.34], [0.191121, 0.680788, 0.701216, -0.091085], [0,0,0,0], [9E9, 9E9, 9E9, 9E9, 9E9, 9E9]];
	VAR robtarget OpenholeUD_2929 := [[489.61, -35.1, 187.73], [0.180649, 0.683642, 0.702684, -0.078962], [0,0,0,0], [9E9, 9E9, 9E9, 9E9, 9E9, 9E9]];
	VAR robtarget OpenholeUD_2930 := [[485.66, -35.1, 187.12], [0.169804, 0.686416, 0.703967, -0.06656], [0,0,0,0], [9E9, 9E9, 9E9, 9E9, 9E9, 9E9]];
	VAR robtarget OpenholeUD_2931 := [[481.71, -35.1, 186.51], [0.158593, 0.689092, 0.705049, -0.053901], [0,0,0,0], [9E9, 9E9, 9E9, 9E9, 9E9, 9E9]];
	VAR robtarget OpenholeUD_2932 := [[477.75, -35.1, 185.89], [0.147029, 0.691652, 0.705916, -0.041015], [0,0,0,0], [9E9, 9E9, 9E9, 9E9, 9E9, 9E9]];
	VAR robtarget OpenholeUD_2933 := [[473.8, -35.1, 185.28], [0.135127, 0.694075, 0.706555, -0.027933], [0,0,0,0], [9E9, 9E9, 9E9, 9E9, 9E9, 9E9]];
	VAR robtarget OpenholeUD_2934 := [[469.85, -35.1, 184.67], [0.122908, 0.696343, 0.706954, -0.01469], [0,0,0,0], [9E9, 9E9, 9E9, 9E9, 9E9, 9E9]];
	VAR robtarget OpenholeUD_2935 := [[465.89, -35.1, 184.06], [0.110397, 0.698436, 0.707106, -0.001325], [0,0,0,0], [9E9, 9E9, 9E9, 9E9, 9E9, 9E9]];
	VAR robtarget OpenholeUD_2936 := [[461.94, -35.1, 183.45], [0.097624, 0.700335, 0.707003, 0.012122], [0,0,0,0], [9E9, 9E9, 9E9, 9E9, 9E9, 9E9]];
	VAR robtarget OpenholeUD_2937 := [[457.99, -35.1, 182.84], [0.084621, 0.702025, 0.706643, 0.025609], [0,0,0,0], [9E9, 9E9, 9E9, 9E9, 9E9, 9E9]];
	VAR robtarget OpenholeUD_2938 := [[454.03, -35.1, 182.23], [0.071424, 0.70349, 0.706025, 0.03909], [0,0,0,0], [9E9, 9E9, 9E9, 9E9, 9E9, 9E9]];
	VAR robtarget OpenholeUD_2939 := [[450.08, -35.1, 181.61], [0.058075, 0.704718, 0.705153, 0.052524], [0,0,0,0], [9E9, 9E9, 9E9, 9E9, 9E9, 9E9]];
	VAR robtarget OpenholeUD_2940 := [[446.13, -35.1, 181], [0.044615, 0.705698, 0.704033, 0.065864], [0,0,0,0], [9E9, 9E9, 9E9, 9E9, 9E9, 9E9]];
	VAR robtarget OpenholeUD_2941 := [[442.17, -35.1, 180.39], [0.031087, 0.706423, 0.702672, 0.079071], [0,0,0,0], [9E9, 9E9, 9E9, 9E9, 9E9, 9E9]];
	VAR robtarget OpenholeUD_2942 := [[438.22, -35.1, 179.78], [0.017537, 0.706889, 0.701083, 0.092103], [0,0,0,0], [9E9, 9E9, 9E9, 9E9, 9E9, 9E9]];
	VAR robtarget OpenholeUD_2943 := [[434.27, -35.1, 179.17], [0.00401, 0.707095, 0.699279, 0.104923], [0,0,0,0], [9E9, 9E9, 9E9, 9E9, 9E9, 9E9]];
	VAR robtarget OpenholeUD_2944 := [[430.32, -35.1, 178.56], [-0.009451, 0.707044, 0.697276, 0.117497], [0,0,0,0], [9E9, 9E9, 9E9, 9E9, 9E9, 9E9]];
	VAR robtarget OpenholeUD_2945 := [[426.36, -35.1, 177.95], [-0.022803, 0.706739, 0.695092, 0.129794], [0,0,0,0], [9E9, 9E9, 9E9, 9E9, 9E9, 9E9]];
	VAR robtarget OpenholeUD_2946 := [[422.41, -35.1, 177.34], [-0.036006, 0.706189, 0.692745, 0.141789], [0,0,0,0], [9E9, 9E9, 9E9, 9E9, 9E9, 9E9]];
	VAR robtarget OpenholeUD_2947 := [[418.46, -35.1, 176.72], [-0.049024, 0.705405, 0.690254, 0.153458], [0,0,0,0], [9E9, 9E9, 9E9, 9E9, 9E9, 9E9]];
	VAR robtarget OpenholeUD_2948 := [[414.5, -35.1, 176.11], [-0.061823, 0.704399, 0.687638, 0.164785], [0,0,0,0], [9E9, 9E9, 9E9, 9E9, 9E9, 9E9]];
	VAR robtarget OpenholeUD_2949 := [[410.55, -35.1, 175.5], [-0.074373, 0.703185, 0.684916, 0.175755], [0,0,0,0], [9E9, 9E9, 9E9, 9E9, 9E9, 9E9]];
	VAR robtarget OpenholeUD_2950 := [[406.6, -35.1, 174.89], [-0.086648, 0.701778, 0.682107, 0.186359], [0,0,0,0], [9E9, 9E9, 9E9, 9E9, 9E9, 9E9]];
	VAR robtarget OpenholeUD_2951 := [[402.64, -35.1, 174.28], [-0.098626, 0.700195, 0.679229, 0.19659], [0,0,0,0], [9E9, 9E9, 9E9, 9E9, 9E9, 9E9]];
	VAR robtarget OpenholeUD_2952 := [[398.69, -35.1, 173.67], [-0.110289, 0.698453, 0.676299, 0.206446], [0,0,0,0], [9E9, 9E9, 9E9, 9E9, 9E9, 9E9]];
	VAR robtarget OpenholeUD_2953 := [[394.74, -35.1, 173.06], [-0.121624, 0.696568, 0.673332, 0.215927], [0,0,0,0], [9E9, 9E9, 9E9, 9E9, 9E9, 9E9]];
	VAR robtarget OpenholeUD_2954 := [[389.32, -35.1, 172.22], [-0.136616, 0.693784, 0.669228, 0.228327], [0,0,0,0], [9E9, 9E9, 9E9, 9E9, 9E9, 9E9]];
	VAR robtarget OpenholeUD_2955 := [[385.32, -35.1, 172.23], [-0.183051, 0.683002, 0.683002, 0.183051], [0,0,0,0], [9E9, 9E9, 9E9, 9E9, 9E9, 9E9]];
	VAR robtarget OpenholeUD_2956 := [[381.32, -35.1, 172.24], [-0.183051, 0.683002, 0.683002, 0.183051], [0,0,0,0], [9E9, 9E9, 9E9, 9E9, 9E9, 9E9]];
	VAR robtarget OpenholeUD_2957 := [[377.32, -35.1, 172.26], [-0.183051, 0.683002, 0.683002, 0.183051], [0,0,0,0], [9E9, 9E9, 9E9, 9E9, 9E9, 9E9]];
	VAR robtarget OpenholeUD_2958 := [[373.32, -35.1, 172.27], [-0.183051, 0.683002, 0.683002, 0.183051], [0,0,0,0], [9E9, 9E9, 9E9, 9E9, 9E9, 9E9]];
	VAR robtarget OpenholeUD_2959 := [[369.32, -35.1, 172.28], [-0.183051, 0.683002, 0.683002, 0.183051], [0,0,0,0], [9E9, 9E9, 9E9, 9E9, 9E9, 9E9]];
	VAR robtarget OpenholeUD_2960 := [[369.32, -35.1, 172.28], [-0.183051, 0.683002, 0.683002, 0.183051], [0,0,0,0], [9E9, 9E9, 9E9, 9E9, 9E9, 9E9]];
	VAR robtarget OpenholeUD_2961 := [[369.32, -33.9, 172.97], [-0.183051, 0.683002, 0.683002, 0.183051], [0,0,0,0], [9E9, 9E9, 9E9, 9E9, 9E9, 9E9]];
	VAR robtarget OpenholeUD_2962 := [[373.32, -33.9, 172.96], [-0.183051, 0.683002, 0.683002, 0.183051], [0,0,0,0], [9E9, 9E9, 9E9, 9E9, 9E9, 9E9]];
	VAR robtarget OpenholeUD_2963 := [[377.32, -33.9, 172.95], [-0.183051, 0.683002, 0.683002, 0.183051], [0,0,0,0], [9E9, 9E9, 9E9, 9E9, 9E9, 9E9]];
	VAR robtarget OpenholeUD_2964 := [[381.32, -33.9, 172.94], [-0.183051, 0.683002, 0.683002, 0.183051], [0,0,0,0], [9E9, 9E9, 9E9, 9E9, 9E9, 9E9]];
	VAR robtarget OpenholeUD_2965 := [[385.32, -33.9, 172.92], [-0.183051, 0.683002, 0.683002, 0.183051], [0,0,0,0], [9E9, 9E9, 9E9, 9E9, 9E9, 9E9]];
	VAR robtarget OpenholeUD_2966 := [[389.32, -33.9, 172.91], [-0.140033, 0.693102, 0.670343, 0.225034], [0,0,0,0], [9E9, 9E9, 9E9, 9E9, 9E9, 9E9]];
	VAR robtarget OpenholeUD_2967 := [[393.28, -33.9, 173.48], [-0.12921, 0.695201, 0.673315, 0.21598], [0,0,0,0], [9E9, 9E9, 9E9, 9E9, 9E9, 9E9]];
	VAR robtarget OpenholeUD_2968 := [[397.24, -33.9, 174.05], [-0.118043, 0.697184, 0.676266, 0.206554], [0,0,0,0], [9E9, 9E9, 9E9, 9E9, 9E9, 9E9]];
	VAR robtarget OpenholeUD_2969 := [[401.2, -33.9, 174.61], [-0.10654, 0.699034, 0.679181, 0.196755], [0,0,0,0], [9E9, 9E9, 9E9, 9E9, 9E9, 9E9]];
	VAR robtarget OpenholeUD_2970 := [[405.16, -33.9, 175.18], [-0.094713, 0.700735, 0.682047, 0.186581], [0,0,0,0], [9E9, 9E9, 9E9, 9E9, 9E9, 9E9]];
	VAR robtarget OpenholeUD_2971 := [[409.12, -33.9, 175.74], [-0.082578, 0.702268, 0.684844, 0.176035], [0,0,0,0], [9E9, 9E9, 9E9, 9E9, 9E9, 9E9]];
	VAR robtarget OpenholeUD_2972 := [[413.08, -33.9, 176.31], [-0.070156, 0.703618, 0.687557, 0.165121], [0,0,0,0], [9E9, 9E9, 9E9, 9E9, 9E9, 9E9]];
	VAR robtarget OpenholeUD_2973 := [[417.04, -33.9, 176.88], [-0.057469, 0.704768, 0.690167, 0.153848], [0,0,0,0], [9E9, 9E9, 9E9, 9E9, 9E9, 9E9]];
	VAR robtarget OpenholeUD_2974 := [[421, -33.9, 177.44], [-0.044546, 0.705702, 0.692655, 0.14223], [0,0,0,0], [9E9, 9E9, 9E9, 9E9, 9E9, 9E9]];
	VAR robtarget OpenholeUD_2975 := [[424.96, -33.9, 178.01], [-0.031419, 0.706408, 0.695001, 0.130283], [0,0,0,0], [9E9, 9E9, 9E9, 9E9, 9E9, 9E9]];
	VAR robtarget OpenholeUD_2976 := [[428.92, -33.9, 178.58], [-0.018124, 0.706874, 0.697187, 0.118029], [0,0,0,0], [9E9, 9E9, 9E9, 9E9, 9E9, 9E9]];
	VAR robtarget OpenholeUD_2977 := [[432.88, -33.9, 179.14], [-0.004699, 0.707091, 0.699193, 0.105494], [0,0,0,0], [9E9, 9E9, 9E9, 9E9, 9E9, 9E9]];
	VAR robtarget OpenholeUD_2978 := [[436.84, -33.9, 179.71], [0.008814, 0.707052, 0.701003, 0.092705], [0,0,0,0], [9E9, 9E9, 9E9, 9E9, 9E9, 9E9]];
	VAR robtarget OpenholeUD_2979 := [[440.8, -33.9, 180.28], [0.022371, 0.706753, 0.702601, 0.079698], [0,0,0,0], [9E9, 9E9, 9E9, 9E9, 9E9, 9E9]];
	VAR robtarget OpenholeUD_2980 := [[444.75, -33.9, 180.84], [0.03593, 0.706193, 0.703972, 0.066509], [0,0,0,0], [9E9, 9E9, 9E9, 9E9, 9E9, 9E9]];
	VAR robtarget OpenholeUD_2981 := [[448.71, -33.9, 181.41], [0.049443, 0.705376, 0.705104, 0.053177], [0,0,0,0], [9E9, 9E9, 9E9, 9E9, 9E9, 9E9]];
	VAR robtarget OpenholeUD_2982 := [[452.67, -33.9, 181.98], [0.062867, 0.704307, 0.705989, 0.039745], [0,0,0,0], [9E9, 9E9, 9E9, 9E9, 9E9, 9E9]];
	VAR robtarget OpenholeUD_2983 := [[456.63, -33.9, 182.54], [0.076159, 0.702993, 0.706619, 0.026256], [0,0,0,0], [9E9, 9E9, 9E9, 9E9, 9E9, 9E9]];
	VAR robtarget OpenholeUD_2984 := [[460.59, -33.9, 183.11], [0.089277, 0.701448, 0.706992, 0.012754], [0,0,0,0], [9E9, 9E9, 9E9, 9E9, 9E9, 9E9]];
	VAR robtarget OpenholeUD_2985 := [[464.55, -33.9, 183.68], [0.102183, 0.699685, 0.707106, -0.000717], [0,0,0,0], [9E9, 9E9, 9E9, 9E9, 9E9, 9E9]];
	VAR robtarget OpenholeUD_2986 := [[468.51, -33.9, 184.24], [0.114842, 0.697719, 0.706966, -0.014114], [0,0,0,0], [9E9, 9E9, 9E9, 9E9, 9E9, 9E9]];
	VAR robtarget OpenholeUD_2987 := [[472.47, -33.9, 184.81], [0.127223, 0.695568, 0.706576, -0.027395], [0,0,0,0], [9E9, 9E9, 9E9, 9E9, 9E9, 9E9]];
	VAR robtarget OpenholeUD_2988 := [[476.43, -33.9, 185.38], [0.139299, 0.69325, 0.705945, -0.040522], [0,0,0,0], [9E9, 9E9, 9E9, 9E9, 9E9, 9E9]];
	VAR robtarget OpenholeUD_2989 := [[480.39, -33.9, 185.94], [0.151047, 0.690786, 0.705083, -0.053459], [0,0,0,0], [9E9, 9E9, 9E9, 9E9, 9E9, 9E9]];
	VAR robtarget OpenholeUD_2990 := [[484.35, -33.9, 186.51], [0.16245, 0.688193, 0.704004, -0.066172], [0,0,0,0], [9E9, 9E9, 9E9, 9E9, 9E9, 9E9]];
	VAR robtarget OpenholeUD_2991 := [[488.31, -33.9, 187.08], [0.173493, 0.685493, 0.702721, -0.078633], [0,0,0,0], [9E9, 9E9, 9E9, 9E9, 9E9, 9E9]];
	VAR robtarget OpenholeUD_2992 := [[492.27, -33.9, 187.64], [0.184165, 0.682703, 0.70125, -0.090818], [0,0,0,0], [9E9, 9E9, 9E9, 9E9, 9E9, 9E9]];
	VAR robtarget OpenholeUD_2993 := [[496.23, -33.9, 188.21], [0.194462, 0.679841, 0.699608, -0.102704], [0,0,0,0], [9E9, 9E9, 9E9, 9E9, 9E9, 9E9]];
	VAR robtarget OpenholeUD_2994 := [[500.19, -33.9, 188.78], [0.204381, 0.676926, 0.697812, -0.114275], [0,0,0,0], [9E9, 9E9, 9E9, 9E9, 9E9, 9E9]];
	VAR robtarget OpenholeUD_2995 := [[504.15, -33.9, 189.34], [0.213921, 0.673972, 0.695877, -0.125517], [0,0,0,0], [9E9, 9E9, 9E9, 9E9, 9E9, 9E9]];
	VAR robtarget OpenholeUD_2996 := [[509.37, -33.9, 190.09], [0.183051, 0.683002, 0.683002, -0.183051], [0,0,0,0], [9E9, 9E9, 9E9, 9E9, 9E9, 9E9]];
	VAR robtarget OpenholeUD_2997 := [[513.37, -33.9, 190.08], [0.183051, 0.683002, 0.683002, -0.183051], [0,0,0,0], [9E9, 9E9, 9E9, 9E9, 9E9, 9E9]];
	VAR robtarget OpenholeUD_2998 := [[517.37, -33.9, 190.07], [0.183051, 0.683002, 0.683002, -0.183051], [0,0,0,0], [9E9, 9E9, 9E9, 9E9, 9E9, 9E9]];
	VAR robtarget OpenholeUD_2999 := [[521.37, -33.9, 190.05], [0.183051, 0.683002, 0.683002, -0.183051], [0,0,0,0], [9E9, 9E9, 9E9, 9E9, 9E9, 9E9]];
	VAR robtarget OpenholeUD_3000 := [[525.37, -33.9, 190.04], [0.183051, 0.683002, 0.683002, -0.183051], [0,0,0,0], [9E9, 9E9, 9E9, 9E9, 9E9, 9E9]];
	VAR robtarget OpenholeUD_3001 := [[529.37, -33.9, 190.03], [0.183051, 0.683002, 0.683002, -0.183051], [0,0,0,0], [9E9, 9E9, 9E9, 9E9, 9E9, 9E9]];
	VAR robtarget OpenholeUD_3002 := [[529.37, -33.9, 190.03], [0.183051, 0.683002, 0.683002, -0.183051], [0,0,0,0], [9E9, 9E9, 9E9, 9E9, 9E9, 9E9]];
	VAR robtarget OpenholeUD_3003 := [[529.37, -32.7, 189.34], [0.183051, 0.683002, 0.683002, -0.183051], [0,0,0,0], [9E9, 9E9, 9E9, 9E9, 9E9, 9E9]];
	VAR robtarget OpenholeUD_3004 := [[525.37, -32.7, 189.35], [0.183051, 0.683002, 0.683002, -0.183051], [0,0,0,0], [9E9, 9E9, 9E9, 9E9, 9E9, 9E9]];
	VAR robtarget OpenholeUD_3005 := [[521.37, -32.7, 189.36], [0.183051, 0.683002, 0.683002, -0.183051], [0,0,0,0], [9E9, 9E9, 9E9, 9E9, 9E9, 9E9]];
	VAR robtarget OpenholeUD_3006 := [[517.37, -32.7, 189.37], [0.183051, 0.683002, 0.683002, -0.183051], [0,0,0,0], [9E9, 9E9, 9E9, 9E9, 9E9, 9E9]];
	VAR robtarget OpenholeUD_3007 := [[513.37, -32.7, 189.39], [0.183051, 0.683002, 0.683002, -0.183051], [0,0,0,0], [9E9, 9E9, 9E9, 9E9, 9E9, 9E9]];
	VAR robtarget OpenholeUD_3008 := [[509.37, -32.7, 189.4], [0.183051, 0.683002, 0.683002, -0.183051], [0,0,0,0], [9E9, 9E9, 9E9, 9E9, 9E9, 9E9]];
	VAR robtarget OpenholeUD_3009 := [[505.41, -32.7, 188.88], [0.213499, 0.674106, 0.694584, -0.132488], [0,0,0,0], [9E9, 9E9, 9E9, 9E9, 9E9, 9E9]];
	VAR robtarget OpenholeUD_3010 := [[501.44, -32.7, 188.35], [0.203996, 0.677042, 0.696608, -0.121398], [0,0,0,0], [9E9, 9E9, 9E9, 9E9, 9E9, 9E9]];
	VAR robtarget OpenholeUD_3011 := [[497.47, -32.7, 187.83], [0.194116, 0.67994, 0.698503, -0.109972], [0,0,0,0], [9E9, 9E9, 9E9, 9E9, 9E9, 9E9]];
	VAR robtarget OpenholeUD_3012 := [[493.51, -32.7, 187.31], [0.183858, 0.682786, 0.700252, -0.098223], [0,0,0,0], [9E9, 9E9, 9E9, 9E9, 9E9, 9E9]];
	VAR robtarget OpenholeUD_3013 := [[489.54, -32.7, 186.79], [0.173224, 0.685561, 0.701837, -0.086166], [0,0,0,0], [9E9, 9E9, 9E9, 9E9, 9E9, 9E9]];
	VAR robtarget OpenholeUD_3014 := [[485.58, -32.7, 186.27], [0.162219, 0.688248, 0.703243, -0.07382], [0,0,0,0], [9E9, 9E9, 9E9, 9E9, 9E9, 9E9]];
	VAR robtarget OpenholeUD_3015 := [[481.61, -32.7, 185.75], [0.150854, 0.690828, 0.704453, -0.061209], [0,0,0,0], [9E9, 9E9, 9E9, 9E9, 9E9, 9E9]];
	VAR robtarget OpenholeUD_3016 := [[477.65, -32.7, 185.22], [0.13914, 0.693282, 0.705451, -0.048361], [0,0,0,0], [9E9, 9E9, 9E9, 9E9, 9E9, 9E9]];
	VAR robtarget OpenholeUD_3017 := [[473.68, -32.7, 184.7], [0.127096, 0.695591, 0.706225, -0.035306], [0,0,0,0], [9E9, 9E9, 9E9, 9E9, 9E9, 9E9]];
	VAR robtarget OpenholeUD_3018 := [[469.71, -32.7, 184.18], [0.114744, 0.697735, 0.706762, -0.022079], [0,0,0,0], [9E9, 9E9, 9E9, 9E9, 9E9, 9E9]];
	VAR robtarget OpenholeUD_3019 := [[465.75, -32.7, 183.66], [0.10211, 0.699695, 0.707053, -0.008717], [0,0,0,0], [9E9, 9E9, 9E9, 9E9, 9E9, 9E9]];
	VAR robtarget OpenholeUD_3020 := [[461.78, -32.7, 183.14], [0.089224, 0.701455, 0.707091, 0.004737], [0,0,0,0], [9E9, 9E9, 9E9, 9E9, 9E9, 9E9]];
	VAR robtarget OpenholeUD_3021 := [[457.82, -32.7, 182.62], [0.076121, 0.702998, 0.706871, 0.018243], [0,0,0,0], [9E9, 9E9, 9E9, 9E9, 9E9, 9E9]];
	VAR robtarget OpenholeUD_3022 := [[453.85, -32.7, 182.09], [0.062839, 0.704309, 0.706393, 0.031755], [0,0,0,0], [9E9, 9E9, 9E9, 9E9, 9E9, 9E9]];
	VAR robtarget OpenholeUD_3023 := [[449.88, -32.7, 181.57], [0.049418, 0.705378, 0.705659, 0.045231], [0,0,0,0], [9E9, 9E9, 9E9, 9E9, 9E9, 9E9]];
	VAR robtarget OpenholeUD_3024 := [[445.92, -32.7, 181.05], [0.035902, 0.706195, 0.704672, 0.058625], [0,0,0,0], [9E9, 9E9, 9E9, 9E9, 9E9, 9E9]];
	VAR robtarget OpenholeUD_3025 := [[441.95, -32.7, 180.53], [0.022334, 0.706754, 0.703442, 0.071895], [0,0,0,0], [9E9, 9E9, 9E9, 9E9, 9E9, 9E9]];
	VAR robtarget OpenholeUD_3026 := [[437.99, -32.7, 180.01], [0.008761, 0.707053, 0.701979, 0.085001], [0,0,0,0], [9E9, 9E9, 9E9, 9E9, 9E9, 9E9]];
	VAR robtarget OpenholeUD_3027 := [[434.02, -32.7, 179.49], [-0.004773, 0.707091, 0.700296, 0.097904], [0,0,0,0], [9E9, 9E9, 9E9, 9E9, 9E9, 9E9]];
	VAR robtarget OpenholeUD_3028 := [[430.06, -32.7, 178.96], [-0.018225, 0.706872, 0.698408, 0.11057], [0,0,0,0], [9E9, 9E9, 9E9, 9E9, 9E9, 9E9]];
	VAR robtarget OpenholeUD_3029 := [[426.09, -32.7, 178.44], [-0.031552, 0.706402, 0.696333, 0.122966], [0,0,0,0], [9E9, 9E9, 9E9, 9E9, 9E9, 9E9]];
	VAR robtarget OpenholeUD_3030 := [[422.12, -32.7, 177.92], [-0.044715, 0.705692, 0.694087, 0.135066], [0,0,0,0], [9E9, 9E9, 9E9, 9E9, 9E9, 9E9]];
	VAR robtarget OpenholeUD_3031 := [[418.16, -32.7, 177.4], [-0.057678, 0.704751, 0.691691, 0.146846], [0,0,0,0], [9E9, 9E9, 9E9, 9E9, 9E9, 9E9]];
	VAR robtarget OpenholeUD_3032 := [[414.19, -32.7, 176.88], [-0.070407, 0.703593, 0.689162, 0.158289], [0,0,0,0], [9E9, 9E9, 9E9, 9E9, 9E9, 9E9]];
	VAR robtarget OpenholeUD_3033 := [[410.23, -32.7, 176.36], [-0.082875, 0.702233, 0.686521, 0.169378], [0,0,0,0], [9E9, 9E9, 9E9, 9E9, 9E9, 9E9]];
	VAR robtarget OpenholeUD_3034 := [[406.26, -32.7, 175.83], [-0.095057, 0.700688, 0.683785, 0.180104], [0,0,0,0], [9E9, 9E9, 9E9, 9E9, 9E9, 9E9]];
	VAR robtarget OpenholeUD_3035 := [[402.29, -32.7, 175.31], [-0.106932, 0.698975, 0.680973, 0.19046], [0,0,0,0], [9E9, 9E9, 9E9, 9E9, 9E9, 9E9]];
	VAR robtarget OpenholeUD_3036 := [[398.33, -32.7, 174.79], [-0.118483, 0.69711, 0.678102, 0.200443], [0,0,0,0], [9E9, 9E9, 9E9, 9E9, 9E9, 9E9]];
	VAR robtarget OpenholeUD_3037 := [[394.36, -32.7, 174.27], [-0.129698, 0.69511, 0.675188, 0.210051], [0,0,0,0], [9E9, 9E9, 9E9, 9E9, 9E9, 9E9]];
	VAR robtarget OpenholeUD_3038 := [[389.32, -32.7, 173.6], [-0.143454, 0.692402, 0.671444, 0.221728], [0,0,0,0], [9E9, 9E9, 9E9, 9E9, 9E9, 9E9]];
	VAR robtarget OpenholeUD_3039 := [[385.32, -32.7, 173.62], [-0.183051, 0.683002, 0.683002, 0.183051], [0,0,0,0], [9E9, 9E9, 9E9, 9E9, 9E9, 9E9]];
	VAR robtarget OpenholeUD_3040 := [[381.32, -32.7, 173.63], [-0.183051, 0.683002, 0.683002, 0.183051], [0,0,0,0], [9E9, 9E9, 9E9, 9E9, 9E9, 9E9]];
	VAR robtarget OpenholeUD_3041 := [[377.32, -32.7, 173.64], [-0.183051, 0.683002, 0.683002, 0.183051], [0,0,0,0], [9E9, 9E9, 9E9, 9E9, 9E9, 9E9]];
	VAR robtarget OpenholeUD_3042 := [[373.32, -32.7, 173.66], [-0.183051, 0.683002, 0.683002, 0.183051], [0,0,0,0], [9E9, 9E9, 9E9, 9E9, 9E9, 9E9]];
	VAR robtarget OpenholeUD_3043 := [[369.32, -32.7, 173.67], [-0.183051, 0.683002, 0.683002, 0.183051], [0,0,0,0], [9E9, 9E9, 9E9, 9E9, 9E9, 9E9]];
	VAR robtarget OpenholeUD_3044 := [[369.32, -32.7, 173.67], [-0.183051, 0.683002, 0.683002, 0.183051], [0,0,0,0], [9E9, 9E9, 9E9, 9E9, 9E9, 9E9]];
	VAR robtarget OpenholeUD_3045 := [[369.32, -31.5, 174.36], [-0.183051, 0.683002, 0.683002, 0.183051], [0,0,0,0], [9E9, 9E9, 9E9, 9E9, 9E9, 9E9]];
	VAR robtarget OpenholeUD_3046 := [[373.32, -31.5, 174.35], [-0.183051, 0.683002, 0.683002, 0.183051], [0,0,0,0], [9E9, 9E9, 9E9, 9E9, 9E9, 9E9]];
	VAR robtarget OpenholeUD_3047 := [[377.32, -31.5, 174.34], [-0.183051, 0.683002, 0.683002, 0.183051], [0,0,0,0], [9E9, 9E9, 9E9, 9E9, 9E9, 9E9]];
	VAR robtarget OpenholeUD_3048 := [[381.32, -31.5, 174.32], [-0.183051, 0.683002, 0.683002, 0.183051], [0,0,0,0], [9E9, 9E9, 9E9, 9E9, 9E9, 9E9]];
	VAR robtarget OpenholeUD_3049 := [[385.32, -31.5, 174.31], [-0.183051, 0.683002, 0.683002, 0.183051], [0,0,0,0], [9E9, 9E9, 9E9, 9E9, 9E9, 9E9]];
	VAR robtarget OpenholeUD_3050 := [[389.32, -31.5, 174.3], [-0.146879, 0.691684, 0.672531, 0.218409], [0,0,0,0], [9E9, 9E9, 9E9, 9E9, 9E9, 9E9]];
	VAR robtarget OpenholeUD_3051 := [[393.3, -31.5, 174.77], [-0.136154, 0.693875, 0.675454, 0.209192], [0,0,0,0], [9E9, 9E9, 9E9, 9E9, 9E9, 9E9]];
	VAR robtarget OpenholeUD_3052 := [[397.27, -31.5, 175.25], [-0.12508, 0.695956, 0.67835, 0.199604], [0,0,0,0], [9E9, 9E9, 9E9, 9E9, 9E9, 9E9]];
	VAR robtarget OpenholeUD_3053 := [[401.24, -31.5, 175.73], [-0.113663, 0.697912, 0.681202, 0.189642], [0,0,0,0], [9E9, 9E9, 9E9, 9E9, 9E9, 9E9]];
	VAR robtarget OpenholeUD_3054 := [[405.21, -31.5, 176.2], [-0.101916, 0.699724, 0.683995, 0.179307], [0,0,0,0], [9E9, 9E9, 9E9, 9E9, 9E9, 9E9]];
	VAR robtarget OpenholeUD_3055 := [[409.18, -31.5, 176.68], [-0.089853, 0.701375, 0.686712, 0.168602], [0,0,0,0], [9E9, 9E9, 9E9, 9E9, 9E9, 9E9]];
	VAR robtarget OpenholeUD_3056 := [[413.15, -31.5, 177.16], [-0.077493, 0.702848, 0.689335, 0.157534], [0,0,0,0], [9E9, 9E9, 9E9, 9E9, 9E9, 9E9]];
	VAR robtarget OpenholeUD_3057 := [[417.12, -31.5, 177.63], [-0.064859, 0.704126, 0.691846, 0.146112], [0,0,0,0], [9E9, 9E9, 9E9, 9E9, 9E9, 9E9]];
	VAR robtarget OpenholeUD_3058 := [[421.1, -31.5, 178.11], [-0.051979, 0.705194, 0.694226, 0.13435], [0,0,0,0], [9E9, 9E9, 9E9, 9E9, 9E9, 9E9]];
	VAR robtarget OpenholeUD_3059 := [[425.07, -31.5, 178.59], [-0.038884, 0.706037, 0.696456, 0.122268], [0,0,0,0], [9E9, 9E9, 9E9, 9E9, 9E9, 9E9]];
	VAR robtarget OpenholeUD_3060 := [[429.04, -31.5, 179.06], [-0.025609, 0.706643, 0.698516, 0.109887], [0,0,0,0], [9E9, 9E9, 9E9, 9E9, 9E9, 9E9]];
	VAR robtarget OpenholeUD_3061 := [[433.01, -31.5, 179.54], [-0.012193, 0.707002, 0.70039, 0.097234], [0,0,0,0], [9E9, 9E9, 9E9, 9E9, 9E9, 9E9]];
	VAR robtarget OpenholeUD_3062 := [[436.98, -31.5, 180.02], [0.001325, 0.707106, 0.702059, 0.084341], [0,0,0,0], [9E9, 9E9, 9E9, 9E9, 9E9, 9E9]];
	VAR robtarget OpenholeUD_3063 := [[440.95, -31.5, 180.49], [0.014899, 0.70695, 0.703509, 0.071242], [0,0,0,0], [9E9, 9E9, 9E9, 9E9, 9E9, 9E9]];
	VAR robtarget OpenholeUD_3064 := [[444.92, -31.5, 180.97], [0.028486, 0.706533, 0.704726, 0.057974], [0,0,0,0], [9E9, 9E9, 9E9, 9E9, 9E9, 9E9]];
	VAR robtarget OpenholeUD_3065 := [[448.9, -31.5, 181.45], [0.04204, 0.705856, 0.7057, 0.044578], [0,0,0,0], [9E9, 9E9, 9E9, 9E9, 9E9, 9E9]];
	VAR robtarget OpenholeUD_3066 := [[452.87, -31.5, 181.92], [0.055517, 0.704924, 0.706423, 0.031097], [0,0,0,0], [9E9, 9E9, 9E9, 9E9, 9E9, 9E9]];
	VAR robtarget OpenholeUD_3067 := [[456.84, -31.5, 182.4], [0.068872, 0.703745, 0.706888, 0.017575], [0,0,0,0], [9E9, 9E9, 9E9, 9E9, 9E9, 9E9]];
	VAR robtarget OpenholeUD_3068 := [[460.81, -31.5, 182.88], [0.082064, 0.702329, 0.707095, 0.004056], [0,0,0,0], [9E9, 9E9, 9E9, 9E9, 9E9, 9E9]];
	VAR robtarget OpenholeUD_3069 := [[464.78, -31.5, 183.35], [0.095053, 0.700689, 0.707044, -0.009416], [0,0,0,0], [9E9, 9E9, 9E9, 9E9, 9E9, 9E9]];
	VAR robtarget OpenholeUD_3070 := [[468.75, -31.5, 183.83], [0.107805, 0.698841, 0.706739, -0.022797], [0,0,0,0], [9E9, 9E9, 9E9, 9E9, 9E9, 9E9]];
	VAR robtarget OpenholeUD_3071 := [[472.73, -31.5, 184.31], [0.120286, 0.696801, 0.706187, -0.036048], [0,0,0,0], [9E9, 9E9, 9E9, 9E9, 9E9, 9E9]];
	VAR robtarget OpenholeUD_3072 := [[476.7, -31.5, 184.78], [0.132469, 0.694588, 0.705398, -0.049129], [0,0,0,0], [9E9, 9E9, 9E9, 9E9, 9E9, 9E9]];
	VAR robtarget OpenholeUD_3073 := [[480.67, -31.5, 185.26], [0.144331, 0.69222, 0.704383, -0.062006], [0,0,0,0], [9E9, 9E9, 9E9, 9E9, 9E9, 9E9]];
	VAR robtarget OpenholeUD_3074 := [[484.64, -31.5, 185.74], [0.155851, 0.689718, 0.703156, -0.074647], [0,0,0,0], [9E9, 9E9, 9E9, 9E9, 9E9, 9E9]];
	VAR robtarget OpenholeUD_3075 := [[488.61, -31.5, 186.21], [0.167016, 0.687099, 0.701731, -0.087024], [0,0,0,0], [9E9, 9E9, 9E9, 9E9, 9E9, 9E9]];
	VAR robtarget OpenholeUD_3076 := [[492.58, -31.5, 186.69], [0.177814, 0.684385, 0.700126, -0.099112], [0,0,0,0], [9E9, 9E9, 9E9, 9E9, 9E9, 9E9]];
	VAR robtarget OpenholeUD_3077 := [[496.55, -31.5, 187.17], [0.188238, 0.681591, 0.698357, -0.110893], [0,0,0,0], [9E9, 9E9, 9E9, 9E9, 9E9, 9E9]];
	VAR robtarget OpenholeUD_3078 := [[500.53, -31.5, 187.64], [0.198286, 0.678736, 0.696441, -0.12235], [0,0,0,0], [9E9, 9E9, 9E9, 9E9, 9E9, 9E9]];
	VAR robtarget OpenholeUD_3079 := [[504.5, -31.5, 188.12], [0.207955, 0.675836, 0.694396, -0.133472], [0,0,0,0], [9E9, 9E9, 9E9, 9E9, 9E9, 9E9]];
	VAR robtarget OpenholeUD_3080 := [[509.37, -31.5, 188.7], [0.183051, 0.683002, 0.683002, -0.183051], [0,0,0,0], [9E9, 9E9, 9E9, 9E9, 9E9, 9E9]];
	VAR robtarget OpenholeUD_3081 := [[513.37, -31.5, 188.69], [0.183051, 0.683002, 0.683002, -0.183051], [0,0,0,0], [9E9, 9E9, 9E9, 9E9, 9E9, 9E9]];
	VAR robtarget OpenholeUD_3082 := [[517.37, -31.5, 188.68], [0.183051, 0.683002, 0.683002, -0.183051], [0,0,0,0], [9E9, 9E9, 9E9, 9E9, 9E9, 9E9]];
	VAR robtarget OpenholeUD_3083 := [[521.37, -31.5, 188.67], [0.183051, 0.683002, 0.683002, -0.183051], [0,0,0,0], [9E9, 9E9, 9E9, 9E9, 9E9, 9E9]];
	VAR robtarget OpenholeUD_3084 := [[529.37, -31.5, 188.64], [0.183051, 0.683002, 0.683002, -0.183051], [0,0,0,0], [9E9, 9E9, 9E9, 9E9, 9E9, 9E9]];
	VAR robtarget OpenholeUD_3085 := [[529.37, -31.5, 188.64], [0.183051, 0.683002, 0.683002, -0.183051], [0,0,0,0], [9E9, 9E9, 9E9, 9E9, 9E9, 9E9]];
	VAR robtarget OpenholeUD_3086 := [[529.37, -30.3, 187.95], [0.183051, 0.683002, 0.683002, -0.183051], [0,0,0,0], [9E9, 9E9, 9E9, 9E9, 9E9, 9E9]];
	VAR robtarget OpenholeUD_3087 := [[525.37, -30.3, 187.96], [0.183051, 0.683002, 0.683002, -0.183051], [0,0,0,0], [9E9, 9E9, 9E9, 9E9, 9E9, 9E9]];
	VAR robtarget OpenholeUD_3088 := [[521.37, -30.3, 187.97], [0.183051, 0.683002, 0.683002, -0.183051], [0,0,0,0], [9E9, 9E9, 9E9, 9E9, 9E9, 9E9]];
	VAR robtarget OpenholeUD_3089 := [[517.37, -30.3, 187.99], [0.183051, 0.683002, 0.683002, -0.183051], [0,0,0,0], [9E9, 9E9, 9E9, 9E9, 9E9, 9E9]];
	VAR robtarget OpenholeUD_3090 := [[509.37, -30.3, 188.01], [0.183051, 0.683002, 0.683002, -0.183051], [0,0,0,0], [9E9, 9E9, 9E9, 9E9, 9E9, 9E9]];
	VAR robtarget OpenholeUD_3091 := [[505.39, -30.3, 187.58], [0.206682, 0.676227, 0.693228, -0.139411], [0,0,0,0], [9E9, 9E9, 9E9, 9E9, 9E9, 9E9]];
	VAR robtarget OpenholeUD_3092 := [[501.41, -30.3, 187.15], [0.197016, 0.679106, 0.695348, -0.128416], [0,0,0,0], [9E9, 9E9, 9E9, 9E9, 9E9, 9E9]];
	VAR robtarget OpenholeUD_3093 := [[497.44, -30.3, 186.72], [0.186974, 0.681939, 0.697347, -0.11708], [0,0,0,0], [9E9, 9E9, 9E9, 9E9, 9E9, 9E9]];
	VAR robtarget OpenholeUD_3094 := [[493.46, -30.3, 186.29], [0.176555, 0.68471, 0.699205, -0.105414], [0,0,0,0], [9E9, 9E9, 9E9, 9E9, 9E9, 9E9]];
	VAR robtarget OpenholeUD_3095 := [[489.48, -30.3, 185.86], [0.165763, 0.687403, 0.700907, -0.093433], [0,0,0,0], [9E9, 9E9, 9E9, 9E9, 9E9, 9E9]];
	VAR robtarget OpenholeUD_3096 := [[485.51, -30.3, 185.42], [0.154604, 0.689998, 0.702434, -0.081154], [0,0,0,0], [9E9, 9E9, 9E9, 9E9, 9E9, 9E9]];
	VAR robtarget OpenholeUD_3097 := [[481.53, -30.3, 184.99], [0.14309, 0.692478, 0.703771, -0.068601], [0,0,0,0], [9E9, 9E9, 9E9, 9E9, 9E9, 9E9]];
	VAR robtarget OpenholeUD_3098 := [[477.55, -30.3, 184.56], [0.131233, 0.694822, 0.704902, -0.0558], [0,0,0,0], [9E9, 9E9, 9E9, 9E9, 9E9, 9E9]];
	VAR robtarget OpenholeUD_3099 := [[473.58, -30.3, 184.13], [0.119055, 0.697012, 0.705811, -0.042782], [0,0,0,0], [9E9, 9E9, 9E9, 9E9, 9E9, 9E9]];
	VAR robtarget OpenholeUD_3100 := [[469.6, -30.3, 183.7], [0.106577, 0.699029, 0.706488, -0.02958], [0,0,0,0], [9E9, 9E9, 9E9, 9E9, 9E9, 9E9]];
	VAR robtarget OpenholeUD_3101 := [[465.62, -30.3, 183.27], [0.093828, 0.700854, 0.70692, -0.016232], [0,0,0,0], [9E9, 9E9, 9E9, 9E9, 9E9, 9E9]];
	VAR robtarget OpenholeUD_3102 := [[461.65, -30.3, 182.84], [0.080838, 0.702471, 0.707101, -0.002779], [0,0,0,0], [9E9, 9E9, 9E9, 9E9, 9E9, 9E9]];
	VAR robtarget OpenholeUD_3103 := [[457.67, -30.3, 182.4], [0.067645, 0.703864, 0.707025, 0.010737], [0,0,0,0], [9E9, 9E9, 9E9, 9E9, 9E9, 9E9]];
	VAR robtarget OpenholeUD_3104 := [[453.69, -30.3, 181.97], [0.054286, 0.70502, 0.70669, 0.024273], [0,0,0,0], [9E9, 9E9, 9E9, 9E9, 9E9, 9E9]];
	VAR robtarget OpenholeUD_3105 := [[449.72, -30.3, 181.54], [0.040804, 0.705928, 0.706097, 0.037784], [0,0,0,0], [9E9, 9E9, 9E9, 9E9, 9E9, 9E9]];
	VAR robtarget OpenholeUD_3106 := [[445.74, -30.3, 181.11], [0.027242, 0.706582, 0.705249, 0.051226], [0,0,0,0], [9E9, 9E9, 9E9, 9E9, 9E9, 9E9]];
	VAR robtarget OpenholeUD_3107 := [[441.76, -30.3, 180.68], [0.013646, 0.706975, 0.704154, 0.064555], [0,0,0,0], [9E9, 9E9, 9E9, 9E9, 9E9, 9E9]];
	VAR robtarget OpenholeUD_3108 := [[437.79, -30.3, 180.25], [0.000059, 0.707107, 0.702821, 0.07773], [0,0,0,0], [9E9, 9E9, 9E9, 9E9, 9E9, 9E9]];
	VAR robtarget OpenholeUD_3109 := [[433.81, -30.3, 179.82], [-0.013472, 0.706978, 0.701264, 0.090713], [0,0,0,0], [9E9, 9E9, 9E9, 9E9, 9E9, 9E9]];
	VAR robtarget OpenholeUD_3110 := [[429.83, -30.3, 179.38], [-0.026904, 0.706595, 0.699496, 0.103467], [0,0,0,0], [9E9, 9E9, 9E9, 9E9, 9E9, 9E9]];
	VAR robtarget OpenholeUD_3111 := [[425.86, -30.3, 178.95], [-0.040195, 0.705963, 0.697534, 0.11596], [0,0,0,0], [9E9, 9E9, 9E9, 9E9, 9E9, 9E9]];
	VAR robtarget OpenholeUD_3112 := [[421.88, -30.3, 178.52], [-0.053308, 0.705094, 0.695395, 0.128164], [0,0,0,0], [9E9, 9E9, 9E9, 9E9, 9E9, 9E9]];
	VAR robtarget OpenholeUD_3113 := [[417.9, -30.3, 178.09], [-0.066207, 0.704, 0.693098, 0.140056], [0,0,0,0], [9E9, 9E9, 9E9, 9E9, 9E9, 9E9]];
	VAR robtarget OpenholeUD_3114 := [[413.93, -30.3, 177.66], [-0.078859, 0.702696, 0.690661, 0.151614], [0,0,0,0], [9E9, 9E9, 9E9, 9E9, 9E9, 9E9]];
	VAR robtarget OpenholeUD_3115 := [[409.95, -30.3, 177.23], [-0.091238, 0.701196, 0.688105, 0.162825], [0,0,0,0], [9E9, 9E9, 9E9, 9E9, 9E9, 9E9]];
	VAR robtarget OpenholeUD_3116 := [[405.97, -30.3, 176.8], [-0.103319, 0.699518, 0.685447, 0.173675], [0,0,0,0], [9E9, 9E9, 9E9, 9E9, 9E9, 9E9]];
	VAR robtarget OpenholeUD_3117 := [[402, -30.3, 176.37], [-0.115084, 0.697679, 0.682705, 0.184158], [0,0,0,0], [9E9, 9E9, 9E9, 9E9, 9E9, 9E9]];
	VAR robtarget OpenholeUD_3118 := [[398.02, -30.3, 175.93], [-0.126517, 0.695696, 0.679897, 0.194269], [0,0,0,0], [9E9, 9E9, 9E9, 9E9, 9E9, 9E9]];
	VAR robtarget OpenholeUD_3119 := [[394.04, -30.3, 175.5], [-0.137607, 0.693588, 0.677039, 0.204006], [0,0,0,0], [9E9, 9E9, 9E9, 9E9, 9E9, 9E9]];
	VAR robtarget OpenholeUD_3120 := [[389.33, -30.3, 174.99], [-0.150308, 0.690947, 0.673603, 0.215078], [0,0,0,0], [9E9, 9E9, 9E9, 9E9, 9E9, 9E9]];
	VAR robtarget OpenholeUD_3121 := [[385.33, -30.3, 175], [-0.183051, 0.683002, 0.683002, 0.183051], [0,0,0,0], [9E9, 9E9, 9E9, 9E9, 9E9, 9E9]];
	VAR robtarget OpenholeUD_3122 := [[381.33, -30.3, 175.02], [-0.183051, 0.683002, 0.683002, 0.183051], [0,0,0,0], [9E9, 9E9, 9E9, 9E9, 9E9, 9E9]];
	VAR robtarget OpenholeUD_3123 := [[377.33, -30.3, 175.03], [-0.183051, 0.683002, 0.683002, 0.183051], [0,0,0,0], [9E9, 9E9, 9E9, 9E9, 9E9, 9E9]];
	VAR robtarget OpenholeUD_3124 := [[373.33, -30.3, 175.04], [-0.183051, 0.683002, 0.683002, 0.183051], [0,0,0,0], [9E9, 9E9, 9E9, 9E9, 9E9, 9E9]];
	VAR robtarget OpenholeUD_3125 := [[369.33, -30.3, 175.05], [-0.183051, 0.683002, 0.683002, 0.183051], [0,0,0,0], [9E9, 9E9, 9E9, 9E9, 9E9, 9E9]];
	VAR robtarget OpenholeUD_3126 := [[369.33, -30.3, 175.05], [-0.183051, 0.683002, 0.683002, 0.183051], [0,0,0,0], [9E9, 9E9, 9E9, 9E9, 9E9, 9E9]];
	VAR robtarget OpenholeUD_3127 := [[369.33, -29.1, 175.75], [-0.183051, 0.683002, 0.683002, 0.183051], [0,0,0,0], [9E9, 9E9, 9E9, 9E9, 9E9, 9E9]];
	VAR robtarget OpenholeUD_3128 := [[373.33, -29.1, 175.73], [-0.183051, 0.683002, 0.683002, 0.183051], [0,0,0,0], [9E9, 9E9, 9E9, 9E9, 9E9, 9E9]];
	VAR robtarget OpenholeUD_3129 := [[377.33, -29.1, 175.72], [-0.183051, 0.683002, 0.683002, 0.183051], [0,0,0,0], [9E9, 9E9, 9E9, 9E9, 9E9, 9E9]];
	VAR robtarget OpenholeUD_3130 := [[381.33, -29.1, 175.71], [-0.183051, 0.683002, 0.683002, 0.183051], [0,0,0,0], [9E9, 9E9, 9E9, 9E9, 9E9, 9E9]];
	VAR robtarget OpenholeUD_3131 := [[385.33, -29.1, 175.7], [-0.183051, 0.683002, 0.683002, 0.183051], [0,0,0,0], [9E9, 9E9, 9E9, 9E9, 9E9, 9E9]];
	VAR robtarget OpenholeUD_3132 := [[389.33, -29.1, 175.68], [-0.153739, 0.690191, 0.674661, 0.211736], [0,0,0,0], [9E9, 9E9, 9E9, 9E9, 9E9, 9E9]];
	VAR robtarget OpenholeUD_3133 := [[393.31, -29.1, 176.07], [-0.143121, 0.692471, 0.677533, 0.202358], [0,0,0,0], [9E9, 9E9, 9E9, 9E9, 9E9, 9E9]];
	VAR robtarget OpenholeUD_3134 := [[397.29, -29.1, 176.46], [-0.132148, 0.694649, 0.680368, 0.192611], [0,0,0,0], [9E9, 9E9, 9E9, 9E9, 9E9, 9E9]];
	VAR robtarget OpenholeUD_3135 := [[401.27, -29.1, 176.84], [-0.120827, 0.696707, 0.683152, 0.18249], [0,0,0,0], [9E9, 9E9, 9E9, 9E9, 9E9, 9E9]];
	VAR robtarget OpenholeUD_3136 := [[405.25, -29.1, 177.23], [-0.109169, 0.698629, 0.685869, 0.171999], [0,0,0,0], [9E9, 9E9, 9E9, 9E9, 9E9, 9E9]];
	VAR robtarget OpenholeUD_3137 := [[409.23, -29.1, 177.61], [-0.097187, 0.700396, 0.688501, 0.161141], [0,0,0,0], [9E9, 9E9, 9E9, 9E9, 9E9, 9E9]];
	VAR robtarget OpenholeUD_3138 := [[413.22, -29.1, 178], [-0.084899, 0.701992, 0.691031, 0.149923], [0,0,0,0], [9E9, 9E9, 9E9, 9E9, 9E9, 9E9]];
	VAR robtarget OpenholeUD_3139 := [[417.2, -29.1, 178.39], [-0.072329, 0.703398, 0.693439, 0.138357], [0,0,0,0], [9E9, 9E9, 9E9, 9E9, 9E9, 9E9]];
	VAR robtarget OpenholeUD_3140 := [[421.18, -29.1, 178.77], [-0.059502, 0.704599, 0.695707, 0.126459], [0,0,0,0], [9E9, 9E9, 9E9, 9E9, 9E9, 9E9]];
	VAR robtarget OpenholeUD_3141 := [[425.16, -29.1, 179.16], [-0.046449, 0.70558, 0.697816, 0.114248], [0,0,0,0], [9E9, 9E9, 9E9, 9E9, 9E9, 9E9]];
	VAR robtarget OpenholeUD_3142 := [[429.14, -29.1, 179.54], [-0.033204, 0.706327, 0.699748, 0.101748], [0,0,0,0], [9E9, 9E9, 9E9, 9E9, 9E9, 9E9]];
	VAR robtarget OpenholeUD_3143 := [[433.12, -29.1, 179.93], [-0.019805, 0.706829, 0.701485, 0.088987], [0,0,0,0], [9E9, 9E9, 9E9, 9E9, 9E9, 9E9]];
	VAR robtarget OpenholeUD_3144 := [[437.1, -29.1, 180.31], [-0.006293, 0.707079, 0.703011, 0.075998], [0,0,0,0], [9E9, 9E9, 9E9, 9E9, 9E9, 9E9]];
	VAR robtarget OpenholeUD_3145 := [[441.09, -29.1, 180.7], [0.007289, 0.707069, 0.704311, 0.062815], [0,0,0,0], [9E9, 9E9, 9E9, 9E9, 9E9, 9E9]];
	VAR robtarget OpenholeUD_3146 := [[445.07, -29.1, 181.09], [0.020897, 0.706798, 0.705374, 0.049478], [0,0,0,0], [9E9, 9E9, 9E9, 9E9, 9E9, 9E9]];
	VAR robtarget OpenholeUD_3147 := [[449.05, -29.1, 181.47], [0.034485, 0.706265, 0.706188, 0.036029], [0,0,0,0], [9E9, 9E9, 9E9, 9E9, 9E9, 9E9]];
	VAR robtarget OpenholeUD_3148 := [[453.03, -29.1, 181.86], [0.048007, 0.705475, 0.706748, 0.022509], [0,0,0,0], [9E9, 9E9, 9E9, 9E9, 9E9, 9E9]];
	VAR robtarget OpenholeUD_3149 := [[457.01, -29.1, 182.24], [0.06142, 0.704434, 0.70705, 0.008965], [0,0,0,0], [9E9, 9E9, 9E9, 9E9, 9E9, 9E9]];
	VAR robtarget OpenholeUD_3150 := [[460.99, -29.1, 182.63], [0.074682, 0.703152, 0.707092, -0.004561], [0,0,0,0], [9E9, 9E9, 9E9, 9E9, 9E9, 9E9]];
	VAR robtarget OpenholeUD_3151 := [[464.97, -29.1, 183.02], [0.087751, 0.701641, 0.706877, -0.018023], [0,0,0,0], [9E9, 9E9, 9E9, 9E9, 9E9, 9E9]];
	VAR robtarget OpenholeUD_3152 := [[468.96, -29.1, 183.4], [0.100592, 0.699915, 0.70641, -0.03138], [0,0,0,0], [9E9, 9E9, 9E9, 9E9, 9E9, 9E9]];
	VAR robtarget OpenholeUD_3153 := [[472.94, -29.1, 183.79], [0.113171, 0.697992, 0.705699, -0.04459], [0,0,0,0], [9E9, 9E9, 9E9, 9E9, 9E9, 9E9]];
	VAR robtarget OpenholeUD_3154 := [[476.92, -29.1, 184.17], [0.12546, 0.695888, 0.704755, -0.057617], [0,0,0,0], [9E9, 9E9, 9E9, 9E9, 9E9, 9E9]];
	VAR robtarget OpenholeUD_3155 := [[480.9, -29.1, 184.56], [0.137434, 0.693622, 0.703591, -0.070426], [0,0,0,0], [9E9, 9E9, 9E9, 9E9, 9E9, 9E9]];
	VAR robtarget OpenholeUD_3156 := [[484.88, -29.1, 184.95], [0.149073, 0.691214, 0.70222, -0.082986], [0,0,0,0], [9E9, 9E9, 9E9, 9E9, 9E9, 9E9]];
	VAR robtarget OpenholeUD_3157 := [[488.86, -29.1, 185.33], [0.16036, 0.688683, 0.700659, -0.095271], [0,0,0,0], [9E9, 9E9, 9E9, 9E9, 9E9, 9E9]];
	VAR robtarget OpenholeUD_3158 := [[492.84, -29.1, 185.72], [0.171285, 0.686048, 0.698925, -0.107257], [0,0,0,0], [9E9, 9E9, 9E9, 9E9, 9E9, 9E9]];
	VAR robtarget OpenholeUD_3159 := [[496.82, -29.1, 186.1], [0.181839, 0.683326, 0.697034, -0.118927], [0,0,0,0], [9E9, 9E9, 9E9, 9E9, 9E9, 9E9]];
	VAR robtarget OpenholeUD_3160 := [[500.81, -29.1, 186.49], [0.192017, 0.680536, 0.695004, -0.130266], [0,0,0,0], [9E9, 9E9, 9E9, 9E9, 9E9, 9E9]];
	VAR robtarget OpenholeUD_3161 := [[504.79, -29.1, 186.88], [0.201819, 0.677694, 0.692853, -0.141261], [0,0,0,0], [9E9, 9E9, 9E9, 9E9, 9E9, 9E9]];
	VAR robtarget OpenholeUD_3162 := [[509.37, -29.1, 187.32], [0.183051, 0.683002, 0.683002, -0.183051], [0,0,0,0], [9E9, 9E9, 9E9, 9E9, 9E9, 9E9]];
	VAR robtarget OpenholeUD_3163 := [[513.37, -29.1, 187.31], [0.183051, 0.683002, 0.683002, -0.183051], [0,0,0,0], [9E9, 9E9, 9E9, 9E9, 9E9, 9E9]];
	VAR robtarget OpenholeUD_3164 := [[517.37, -29.1, 187.29], [0.183051, 0.683002, 0.683002, -0.183051], [0,0,0,0], [9E9, 9E9, 9E9, 9E9, 9E9, 9E9]];
	VAR robtarget OpenholeUD_3165 := [[521.37, -29.1, 187.28], [0.183051, 0.683002, 0.683002, -0.183051], [0,0,0,0], [9E9, 9E9, 9E9, 9E9, 9E9, 9E9]];
	VAR robtarget OpenholeUD_3166 := [[529.37, -29.1, 187.26], [0.183051, 0.683002, 0.683002, -0.183051], [0,0,0,0], [9E9, 9E9, 9E9, 9E9, 9E9, 9E9]];
	VAR robtarget OpenholeUD_3167 := [[529.37, -29.1, 187.26], [0.183051, 0.683002, 0.683002, -0.183051], [0,0,0,0], [9E9, 9E9, 9E9, 9E9, 9E9, 9E9]];
	VAR robtarget OpenholeUD_3168 := [[529.36, -27.9, 186.56], [0.183051, 0.683002, 0.683002, -0.183051], [0,0,0,0], [9E9, 9E9, 9E9, 9E9, 9E9, 9E9]];
	VAR robtarget OpenholeUD_3169 := [[525.36, -27.9, 186.58], [0.183051, 0.683002, 0.683002, -0.183051], [0,0,0,0], [9E9, 9E9, 9E9, 9E9, 9E9, 9E9]];
	VAR robtarget OpenholeUD_3170 := [[521.36, -27.9, 186.59], [0.183051, 0.683002, 0.683002, -0.183051], [0,0,0,0], [9E9, 9E9, 9E9, 9E9, 9E9, 9E9]];
	VAR robtarget OpenholeUD_3171 := [[517.36, -27.9, 186.6], [0.183051, 0.683002, 0.683002, -0.183051], [0,0,0,0], [9E9, 9E9, 9E9, 9E9, 9E9, 9E9]];
	VAR robtarget OpenholeUD_3172 := [[509.36, -27.9, 186.63], [0.183051, 0.683002, 0.683002, -0.183051], [0,0,0,0], [9E9, 9E9, 9E9, 9E9, 9E9, 9E9]];
	VAR robtarget OpenholeUD_3173 := [[505.38, -27.9, 186.29], [0.19982, 0.678286, 0.691795, -0.146353], [0,0,0,0], [9E9, 9E9, 9E9, 9E9, 9E9, 9E9]];
	VAR robtarget OpenholeUD_3174 := [[501.39, -27.9, 185.95], [0.189995, 0.681103, 0.69401, -0.135463], [0,0,0,0], [9E9, 9E9, 9E9, 9E9, 9E9, 9E9]];
	VAR robtarget OpenholeUD_3175 := [[497.41, -27.9, 185.61], [0.179795, 0.683867, 0.696109, -0.124226], [0,0,0,0], [9E9, 9E9, 9E9, 9E9, 9E9, 9E9]];
	VAR robtarget OpenholeUD_3176 := [[493.42, -27.9, 185.26], [0.16922, 0.68656, 0.698076, -0.112652], [0,0,0,0], [9E9, 9E9, 9E9, 9E9, 9E9, 9E9]];
	VAR robtarget OpenholeUD_3177 := [[489.44, -27.9, 184.92], [0.158275, 0.689166, 0.699892, -0.100756], [0,0,0,0], [9E9, 9E9, 9E9, 9E9, 9E9, 9E9]];
	VAR robtarget OpenholeUD_3178 := [[485.45, -27.9, 184.58], [0.146967, 0.691665, 0.70154, -0.088554], [0,0,0,0], [9E9, 9E9, 9E9, 9E9, 9E9, 9E9]];
	VAR robtarget OpenholeUD_3179 := [[481.46, -27.9, 184.24], [0.13531, 0.69404, 0.703003, -0.076069], [0,0,0,0], [9E9, 9E9, 9E9, 9E9, 9E9, 9E9]];
	VAR robtarget OpenholeUD_3180 := [[477.48, -27.9, 183.9], [0.123318, 0.696271, 0.704266, -0.063325], [0,0,0,0], [9E9, 9E9, 9E9, 9E9, 9E9, 9E9]];
	VAR robtarget OpenholeUD_3181 := [[473.49, -27.9, 183.56], [0.111012, 0.698338, 0.705312, -0.050354], [0,0,0,0], [9E9, 9E9, 9E9, 9E9, 9E9, 9E9]];
	VAR robtarget OpenholeUD_3182 := [[469.51, -27.9, 183.22], [0.098417, 0.700224, 0.706128, -0.037187], [0,0,0,0], [9E9, 9E9, 9E9, 9E9, 9E9, 9E9]];
	VAR robtarget OpenholeUD_3183 := [[465.52, -27.9, 182.88], [0.085561, 0.701911, 0.706704, -0.023862], [0,0,0,0], [9E9, 9E9, 9E9, 9E9, 9E9, 9E9]];
	VAR robtarget OpenholeUD_3184 := [[461.54, -27.9, 182.54], [0.072478, 0.703383, 0.70703, -0.01042], [0,0,0,0], [9E9, 9E9, 9E9, 9E9, 9E9, 9E9]];
	VAR robtarget OpenholeUD_3185 := [[457.55, -27.9, 182.2], [0.059204, 0.704624, 0.7071, 0.003099], [0,0,0,0], [9E9, 9E9, 9E9, 9E9, 9E9, 9E9]];
	VAR robtarget OpenholeUD_3186 := [[453.57, -27.9, 181.86], [0.045779, 0.705623, 0.706911, 0.016651], [0,0,0,0], [9E9, 9E9, 9E9, 9E9, 9E9, 9E9]];
	VAR robtarget OpenholeUD_3187 := [[449.58, -27.9, 181.52], [0.032246, 0.706371, 0.706462, 0.03019], [0,0,0,0], [9E9, 9E9, 9E9, 9E9, 9E9, 9E9]];
	VAR robtarget OpenholeUD_3188 := [[445.6, -27.9, 181.18], [0.018649, 0.706861, 0.705757, 0.043672], [0,0,0,0], [9E9, 9E9, 9E9, 9E9, 9E9, 9E9]];
	VAR robtarget OpenholeUD_3189 := [[441.61, -27.9, 180.84], [0.005033, 0.707089, 0.704801, 0.057055], [0,0,0,0], [9E9, 9E9, 9E9, 9E9, 9E9, 9E9]];
	VAR robtarget OpenholeUD_3190 := [[437.62, -27.9, 180.5], [-0.008556, 0.707055, 0.703604, 0.070294], [0,0,0,0], [9E9, 9E9, 9E9, 9E9, 9E9, 9E9]];
	VAR robtarget OpenholeUD_3191 := [[433.64, -27.9, 180.16], [-0.022073, 0.706762, 0.702177, 0.083352], [0,0,0,0], [9E9, 9E9, 9E9, 9E9, 9E9, 9E9]];
	VAR robtarget OpenholeUD_3192 := [[429.65, -27.9, 179.82], [-0.035476, 0.706216, 0.700533, 0.096192], [0,0,0,0], [9E9, 9E9, 9E9, 9E9, 9E9, 9E9]];
	VAR robtarget OpenholeUD_3193 := [[425.67, -27.9, 179.48], [-0.048723, 0.705426, 0.698689, 0.10878], [0,0,0,0], [9E9, 9E9, 9E9, 9E9, 9E9, 9E9]];
	VAR robtarget OpenholeUD_3194 := [[421.68, -27.9, 179.14], [-0.061777, 0.704403, 0.696662, 0.121087], [0,0,0,0], [9E9, 9E9, 9E9, 9E9, 9E9, 9E9]];
	VAR robtarget OpenholeUD_3195 := [[417.7, -27.9, 178.8], [-0.074602, 0.70316, 0.694469, 0.133088], [0,0,0,0], [9E9, 9E9, 9E9, 9E9, 9E9, 9E9]];
	VAR robtarget OpenholeUD_3196 := [[413.71, -27.9, 178.46], [-0.08717, 0.701713, 0.69213, 0.144763], [0,0,0,0], [9E9, 9E9, 9E9, 9E9, 9E9, 9E9]];
	VAR robtarget OpenholeUD_3197 := [[409.73, -27.9, 178.12], [-0.099452, 0.700078, 0.689663, 0.156094], [0,0,0,0], [9E9, 9E9, 9E9, 9E9, 9E9, 9E9]];
	VAR robtarget OpenholeUD_3198 := [[405.74, -27.9, 177.78], [-0.111427, 0.698272, 0.687086, 0.16707], [0,0,0,0], [9E9, 9E9, 9E9, 9E9, 9E9, 9E9]];
	VAR robtarget OpenholeUD_3199 := [[401.75, -27.9, 177.44], [-0.123076, 0.696313, 0.684419, 0.177681], [0,0,0,0], [9E9, 9E9, 9E9, 9E9, 9E9, 9E9]];
	VAR robtarget OpenholeUD_3200 := [[397.77, -27.9, 177.1], [-0.134387, 0.694219, 0.681678, 0.187922], [0,0,0,0], [9E9, 9E9, 9E9, 9E9, 9E9, 9E9]];
	VAR robtarget OpenholeUD_3201 := [[393.78, -27.9, 176.76], [-0.145347, 0.692007, 0.67888, 0.197792], [0,0,0,0], [9E9, 9E9, 9E9, 9E9, 9E9, 9E9]];
	VAR robtarget OpenholeUD_3202 := [[389.33, -27.9, 176.38], [-0.157173, 0.689418, 0.675705, 0.208383], [0,0,0,0], [9E9, 9E9, 9E9, 9E9, 9E9, 9E9]];
	VAR robtarget OpenholeUD_3203 := [[385.33, -27.9, 176.39], [-0.183051, 0.683002, 0.683002, 0.183051], [0,0,0,0], [9E9, 9E9, 9E9, 9E9, 9E9, 9E9]];
	VAR robtarget OpenholeUD_3204 := [[381.33, -27.9, 176.4], [-0.183051, 0.683002, 0.683002, 0.183051], [0,0,0,0], [9E9, 9E9, 9E9, 9E9, 9E9, 9E9]];
	VAR robtarget OpenholeUD_3205 := [[377.33, -27.9, 176.41], [-0.183051, 0.683002, 0.683002, 0.183051], [0,0,0,0], [9E9, 9E9, 9E9, 9E9, 9E9, 9E9]];
	VAR robtarget OpenholeUD_3206 := [[373.33, -27.9, 176.43], [-0.183051, 0.683002, 0.683002, 0.183051], [0,0,0,0], [9E9, 9E9, 9E9, 9E9, 9E9, 9E9]];
	VAR robtarget OpenholeUD_3207 := [[369.33, -27.9, 176.44], [-0.183051, 0.683002, 0.683002, 0.183051], [0,0,0,0], [9E9, 9E9, 9E9, 9E9, 9E9, 9E9]];
	VAR robtarget OpenholeUD_3208 := [[369.33, -27.9, 176.44], [-0.183051, 0.683002, 0.683002, 0.183051], [0,0,0,0], [9E9, 9E9, 9E9, 9E9, 9E9, 9E9]];
	VAR robtarget OpenholeUD_3209 := [[369.33, -26.7, 177.13], [-0.183051, 0.683002, 0.683002, 0.183051], [0,0,0,0], [9E9, 9E9, 9E9, 9E9, 9E9, 9E9]];
	VAR robtarget OpenholeUD_3210 := [[373.33, -26.7, 177.12], [-0.183051, 0.683002, 0.683002, 0.183051], [0,0,0,0], [9E9, 9E9, 9E9, 9E9, 9E9, 9E9]];
	VAR robtarget OpenholeUD_3211 := [[377.33, -26.7, 177.11], [-0.183051, 0.683002, 0.683002, 0.183051], [0,0,0,0], [9E9, 9E9, 9E9, 9E9, 9E9, 9E9]];
	VAR robtarget OpenholeUD_3212 := [[381.33, -26.7, 177.1], [-0.183051, 0.683002, 0.683002, 0.183051], [0,0,0,0], [9E9, 9E9, 9E9, 9E9, 9E9, 9E9]];
	VAR robtarget OpenholeUD_3213 := [[385.33, -26.7, 177.08], [-0.183051, 0.683002, 0.683002, 0.183051], [0,0,0,0], [9E9, 9E9, 9E9, 9E9, 9E9, 9E9]];
	VAR robtarget OpenholeUD_3214 := [[389.33, -26.7, 177.07], [-0.160608, 0.688626, 0.676733, 0.205019], [0,0,0,0], [9E9, 9E9, 9E9, 9E9, 9E9, 9E9]];
	VAR robtarget OpenholeUD_3215 := [[393.32, -26.7, 177.36], [-0.150104, 0.690991, 0.679548, 0.195485], [0,0,0,0], [9E9, 9E9, 9E9, 9E9, 9E9, 9E9]];
	VAR robtarget OpenholeUD_3216 := [[397.31, -26.7, 177.66], [-0.13924, 0.693262, 0.682319, 0.185582], [0,0,0,0], [9E9, 9E9, 9E9, 9E9, 9E9, 9E9]];
	VAR robtarget OpenholeUD_3217 := [[401.3, -26.7, 177.95], [-0.128024, 0.695421, 0.685031, 0.175307], [0,0,0,0], [9E9, 9E9, 9E9, 9E9, 9E9, 9E9]];
	VAR robtarget OpenholeUD_3218 := [[405.29, -26.7, 178.25], [-0.116464, 0.69745, 0.687667, 0.164664], [0,0,0,0], [9E9, 9E9, 9E9, 9E9, 9E9, 9E9]];
	VAR robtarget OpenholeUD_3219 := [[409.28, -26.7, 178.54], [-0.104573, 0.699331, 0.69021, 0.153657], [0,0,0,0], [9E9, 9E9, 9E9, 9E9, 9E9, 9E9]];
	VAR robtarget OpenholeUD_3220 := [[413.27, -26.7, 178.84], [-0.092368, 0.701048, 0.692641, 0.142297], [0,0,0,0], [9E9, 9E9, 9E9, 9E9, 9E9, 9E9]];
	VAR robtarget OpenholeUD_3221 := [[417.26, -26.7, 179.13], [-0.079871, 0.702581, 0.694943, 0.130594], [0,0,0,0], [9E9, 9E9, 9E9, 9E9, 9E9, 9E9]];
	VAR robtarget OpenholeUD_3222 := [[421.25, -26.7, 179.43], [-0.067107, 0.703915, 0.697095, 0.118566], [0,0,0,0], [9E9, 9E9, 9E9, 9E9, 9E9, 9E9]];
	VAR robtarget OpenholeUD_3223 := [[425.23, -26.7, 179.72], [-0.054105, 0.705034, 0.699081, 0.106234], [0,0,0,0], [9E9, 9E9, 9E9, 9E9, 9E9, 9E9]];
	VAR robtarget OpenholeUD_3224 := [[429.22, -26.7, 180.02], [-0.0409, 0.705923, 0.700881, 0.093623], [0,0,0,0], [9E9, 9E9, 9E9, 9E9, 9E9, 9E9]];
	VAR robtarget OpenholeUD_3225 := [[433.21, -26.7, 180.31], [-0.027529, 0.706571, 0.702479, 0.080763], [0,0,0,0], [9E9, 9E9, 9E9, 9E9, 9E9, 9E9]];
	VAR robtarget OpenholeUD_3226 := [[437.2, -26.7, 180.6], [-0.014031, 0.706968, 0.70386, 0.067687], [0,0,0,0], [9E9, 9E9, 9E9, 9E9, 9E9, 9E9]];
	VAR robtarget OpenholeUD_3227 := [[441.19, -26.7, 180.9], [-0.00045, 0.707107, 0.705009, 0.054431], [0,0,0,0], [9E9, 9E9, 9E9, 9E9, 9E9, 9E9]];
	VAR robtarget OpenholeUD_3228 := [[445.18, -26.7, 181.19], [0.01317, 0.706984, 0.705915, 0.041035], [0,0,0,0], [9E9, 9E9, 9E9, 9E9, 9E9, 9E9]];
	VAR robtarget OpenholeUD_3229 := [[449.17, -26.7, 181.49], [0.026784, 0.706599, 0.70657, 0.027541], [0,0,0,0], [9E9, 9E9, 9E9, 9E9, 9E9, 9E9]];
	VAR robtarget OpenholeUD_3230 := [[453.16, -26.7, 181.78], [0.040345, 0.705955, 0.706968, 0.013993], [0,0,0,0], [9E9, 9E9, 9E9, 9E9, 9E9, 9E9]];
	VAR robtarget OpenholeUD_3231 := [[457.15, -26.7, 182.08], [0.05381, 0.705056, 0.707107, 0.000436], [0,0,0,0], [9E9, 9E9, 9E9, 9E9, 9E9, 9E9]];
	VAR robtarget OpenholeUD_3232 := [[461.14, -26.7, 182.37], [0.067135, 0.703913, 0.706986, -0.013086], [0,0,0,0], [9E9, 9E9, 9E9, 9E9, 9E9, 9E9]];
	VAR robtarget OpenholeUD_3233 := [[465.13, -26.7, 182.67], [0.08028, 0.702535, 0.706609, -0.026529], [0,0,0,0], [9E9, 9E9, 9E9, 9E9, 9E9, 9E9]];
	VAR robtarget OpenholeUD_3234 := [[469.12, -26.7, 182.96], [0.093207, 0.700937, 0.705983, -0.039852], [0,0,0,0], [9E9, 9E9, 9E9, 9E9, 9E9, 9E9]];
	VAR robtarget OpenholeUD_3235 := [[473.1, -26.7, 183.26], [0.105881, 0.699135, 0.705117, -0.053013], [0,0,0,0], [9E9, 9E9, 9E9, 9E9, 9E9, 9E9]];
	VAR robtarget OpenholeUD_3236 := [[477.09, -26.7, 183.55], [0.118274, 0.697145, 0.704022, -0.065977], [0,0,0,0], [9E9, 9E9, 9E9, 9E9, 9E9, 9E9]];
	VAR robtarget OpenholeUD_3237 := [[481.08, -26.7, 183.84], [0.13036, 0.694987, 0.702712, -0.07871], [0,0,0,0], [9E9, 9E9, 9E9, 9E9, 9E9, 9E9]];
	VAR robtarget OpenholeUD_3238 := [[485.07, -26.7, 184.14], [0.142116, 0.692678, 0.701203, -0.091182], [0,0,0,0], [9E9, 9E9, 9E9, 9E9, 9E9, 9E9]];
	VAR robtarget OpenholeUD_3239 := [[489.06, -26.7, 184.43], [0.153527, 0.690239, 0.699511, -0.103369], [0,0,0,0], [9E9, 9E9, 9E9, 9E9, 9E9, 9E9]];
	VAR robtarget OpenholeUD_3240 := [[493.05, -26.7, 184.73], [0.164578, 0.687687, 0.697652, -0.115247], [0,0,0,0], [9E9, 9E9, 9E9, 9E9, 9E9, 9E9]];
	VAR robtarget OpenholeUD_3241 := [[497.04, -26.7, 185.02], [0.175263, 0.685042, 0.695645, -0.126801], [0,0,0,0], [9E9, 9E9, 9E9, 9E9, 9E9, 9E9]];
	VAR robtarget OpenholeUD_3242 := [[501.03, -26.7, 185.32], [0.185574, 0.682321, 0.693507, -0.138016], [0,0,0,0], [9E9, 9E9, 9E9, 9E9, 9E9, 9E9]];
	VAR robtarget OpenholeUD_3243 := [[505.02, -26.7, 185.61], [0.195511, 0.679541, 0.691255, -0.148882], [0,0,0,0], [9E9, 9E9, 9E9, 9E9, 9E9, 9E9]];
	VAR robtarget OpenholeUD_3244 := [[509.36, -26.7, 185.93], [0.183051, 0.683002, 0.683002, -0.183051], [0,0,0,0], [9E9, 9E9, 9E9, 9E9, 9E9, 9E9]];
	VAR robtarget OpenholeUD_3245 := [[513.36, -26.7, 185.92], [0.183051, 0.683002, 0.683002, -0.183051], [0,0,0,0], [9E9, 9E9, 9E9, 9E9, 9E9, 9E9]];
	VAR robtarget OpenholeUD_3246 := [[517.36, -26.7, 185.91], [0.183051, 0.683002, 0.683002, -0.183051], [0,0,0,0], [9E9, 9E9, 9E9, 9E9, 9E9, 9E9]];
	VAR robtarget OpenholeUD_3247 := [[521.36, -26.7, 185.9], [0.183051, 0.683002, 0.683002, -0.183051], [0,0,0,0], [9E9, 9E9, 9E9, 9E9, 9E9, 9E9]];
	VAR robtarget OpenholeUD_3248 := [[525.36, -26.7, 185.88], [0.183051, 0.683002, 0.683002, -0.183051], [0,0,0,0], [9E9, 9E9, 9E9, 9E9, 9E9, 9E9]];
	VAR robtarget OpenholeUD_3249 := [[529.36, -26.7, 185.87], [0.183051, 0.683002, 0.683002, -0.183051], [0,0,0,0], [9E9, 9E9, 9E9, 9E9, 9E9, 9E9]];
	VAR robtarget OpenholeUD_3250 := [[529.36, -26.7, 185.87], [0.183051, 0.683002, 0.683002, -0.183051], [0,0,0,0], [9E9, 9E9, 9E9, 9E9, 9E9, 9E9]];
	VAR robtarget OpenholeUD_3251 := [[529.36, -25.5, 185.18], [0.183051, 0.683002, 0.683002, -0.183051], [0,0,0,0], [9E9, 9E9, 9E9, 9E9, 9E9, 9E9]];
	VAR robtarget OpenholeUD_3252 := [[525.36, -25.5, 185.19], [0.183051, 0.683002, 0.683002, -0.183051], [0,0,0,0], [9E9, 9E9, 9E9, 9E9, 9E9, 9E9]];
	VAR robtarget OpenholeUD_3253 := [[521.36, -25.5, 185.2], [0.183051, 0.683002, 0.683002, -0.183051], [0,0,0,0], [9E9, 9E9, 9E9, 9E9, 9E9, 9E9]];
	VAR robtarget OpenholeUD_3254 := [[517.36, -25.5, 185.21], [0.183051, 0.683002, 0.683002, -0.183051], [0,0,0,0], [9E9, 9E9, 9E9, 9E9, 9E9, 9E9]];
	VAR robtarget OpenholeUD_3255 := [[513.36, -25.5, 185.23], [0.183051, 0.683002, 0.683002, -0.183051], [0,0,0,0], [9E9, 9E9, 9E9, 9E9, 9E9, 9E9]];
	VAR robtarget OpenholeUD_3256 := [[509.36, -25.5, 185.24], [0.183051, 0.683002, 0.683002, -0.183051], [0,0,0,0], [9E9, 9E9, 9E9, 9E9, 9E9, 9E9]];
	VAR robtarget OpenholeUD_3257 := [[505.37, -25.5, 184.99], [0.19292, 0.680281, 0.690287, -0.15331], [0,0,0,0], [9E9, 9E9, 9E9, 9E9, 9E9, 9E9]];
	VAR robtarget OpenholeUD_3258 := [[501.37, -25.5, 184.74], [0.18294, 0.683032, 0.692593, -0.142531], [0,0,0,0], [9E9, 9E9, 9E9, 9E9, 9E9, 9E9]];
	VAR robtarget OpenholeUD_3259 := [[497.38, -25.5, 184.49], [0.172586, 0.685722, 0.69479, -0.131402], [0,0,0,0], [9E9, 9E9, 9E9, 9E9, 9E9, 9E9]];
	VAR robtarget OpenholeUD_3260 := [[493.39, -25.5, 184.25], [0.16186, 0.688332, 0.696862, -0.11993], [0,0,0,0], [9E9, 9E9, 9E9, 9E9, 9E9, 9E9]];
	VAR robtarget OpenholeUD_3261 := [[489.4, -25.5, 184], [0.150767, 0.690847, 0.698791, -0.108128], [0,0,0,0], [9E9, 9E9, 9E9, 9E9, 9E9, 9E9]];
	VAR robtarget OpenholeUD_3262 := [[485.41, -25.5, 183.75], [0.139318, 0.693246, 0.700558, -0.096012], [0,0,0,0], [9E9, 9E9, 9E9, 9E9, 9E9, 9E9]];
	VAR robtarget OpenholeUD_3263 := [[481.41, -25.5, 183.5], [0.127524, 0.695512, 0.702147, -0.083604], [0,0,0,0], [9E9, 9E9, 9E9, 9E9, 9E9, 9E9]];
	VAR robtarget OpenholeUD_3264 := [[477.42, -25.5, 183.25], [0.115404, 0.697626, 0.70354, -0.070928], [0,0,0,0], [9E9, 9E9, 9E9, 9E9, 9E9, 9E9]];
	VAR robtarget OpenholeUD_3265 := [[473.43, -25.5, 183], [0.102979, 0.699568, 0.704723, -0.058013], [0,0,0,0], [9E9, 9E9, 9E9, 9E9, 9E9, 9E9]];
	VAR robtarget OpenholeUD_3266 := [[469.44, -25.5, 182.75], [0.090275, 0.70132, 0.70568, -0.044891], [0,0,0,0], [9E9, 9E9, 9E9, 9E9, 9E9, 9E9]];
	VAR robtarget OpenholeUD_3267 := [[465.44, -25.5, 182.5], [0.077322, 0.702867, 0.7064, -0.031599], [0,0,0,0], [9E9, 9E9, 9E9, 9E9, 9E9, 9E9]];
	VAR robtarget OpenholeUD_3268 := [[461.45, -25.5, 182.26], [0.064154, 0.704191, 0.706873, -0.018176], [0,0,0,0], [9E9, 9E9, 9E9, 9E9, 9E9, 9E9]];
	VAR robtarget OpenholeUD_3269 := [[457.46, -25.5, 182.01], [0.050809, 0.705279, 0.707091, -0.004663], [0,0,0,0], [9E9, 9E9, 9E9, 9E9, 9E9, 9E9]];
	VAR robtarget OpenholeUD_3270 := [[453.47, -25.5, 181.76], [0.037328, 0.706121, 0.707051, 0.008895], [0,0,0,0], [9E9, 9E9, 9E9, 9E9, 9E9, 9E9]];
	VAR robtarget OpenholeUD_3271 := [[449.47, -25.5, 181.51], [0.023754, 0.706708, 0.70675, 0.022455], [0,0,0,0], [9E9, 9E9, 9E9, 9E9, 9E9, 9E9]];
	VAR robtarget OpenholeUD_3272 := [[445.48, -25.5, 181.26], [0.010132, 0.707034, 0.706191, 0.035971], [0,0,0,0], [9E9, 9E9, 9E9, 9E9, 9E9, 9E9]];
	VAR robtarget OpenholeUD_3273 := [[441.49, -25.5, 181.01], [-0.003492, 0.707098, 0.705379, 0.0494], [0,0,0,0], [9E9, 9E9, 9E9, 9E9, 9E9, 9E9]];
	VAR robtarget OpenholeUD_3274 := [[437.5, -25.5, 180.76], [-0.017074, 0.706901, 0.704322, 0.062699], [0,0,0,0], [9E9, 9E9, 9E9, 9E9, 9E9, 9E9]];
	VAR robtarget OpenholeUD_3275 := [[433.51, -25.5, 180.51], [-0.030568, 0.706446, 0.703029, 0.075828], [0,0,0,0], [9E9, 9E9, 9E9, 9E9, 9E9, 9E9]];
	VAR robtarget OpenholeUD_3276 := [[429.51, -25.5, 180.27], [-0.043932, 0.705741, 0.701515, 0.088749], [0,0,0,0], [9E9, 9E9, 9E9, 9E9, 9E9, 9E9]];
	VAR robtarget OpenholeUD_3277 := [[425.52, -25.5, 180.02], [-0.057125, 0.704796, 0.699794, 0.101428], [0,0,0,0], [9E9, 9E9, 9E9, 9E9, 9E9, 9E9]];
	VAR robtarget OpenholeUD_3278 := [[421.53, -25.5, 179.77], [-0.070111, 0.703622, 0.697884, 0.113836], [0,0,0,0], [9E9, 9E9, 9E9, 9E9, 9E9, 9E9]];
	VAR robtarget OpenholeUD_3279 := [[417.54, -25.5, 179.52], [-0.082857, 0.702236, 0.6958, 0.125945], [0,0,0,0], [9E9, 9E9, 9E9, 9E9, 9E9, 9E9]];
	VAR robtarget OpenholeUD_3280 := [[413.54, -25.5, 179.27], [-0.095332, 0.700651, 0.693563, 0.137735], [0,0,0,0], [9E9, 9E9, 9E9, 9E9, 9E9, 9E9]];
	VAR robtarget OpenholeUD_3281 := [[409.55, -25.5, 179.02], [-0.107512, 0.698886, 0.69119, 0.149188], [0,0,0,0], [9E9, 9E9, 9E9, 9E9, 9E9, 9E9]];
	VAR robtarget OpenholeUD_3282 := [[405.56, -25.5, 178.77], [-0.119375, 0.696957, 0.6887, 0.160289], [0,0,0,0], [9E9, 9E9, 9E9, 9E9, 9E9, 9E9]];
	VAR robtarget OpenholeUD_3283 := [[401.57, -25.5, 178.53], [-0.130904, 0.694884, 0.686112, 0.171029], [0,0,0,0], [9E9, 9E9, 9E9, 9E9, 9E9, 9E9]];
	VAR robtarget OpenholeUD_3284 := [[397.58, -25.5, 178.28], [-0.142088, 0.692684, 0.683442, 0.181403], [0,0,0,0], [9E9, 9E9, 9E9, 9E9, 9E9, 9E9]];
	VAR robtarget OpenholeUD_3285 := [[393.58, -25.5, 178.03], [-0.152916, 0.690374, 0.680708, 0.191406], [0,0,0,0], [9E9, 9E9, 9E9, 9E9, 9E9, 9E9]];
	VAR robtarget OpenholeUD_3286 := [[389.33, -25.5, 177.76], [-0.164043, 0.687815, 0.677745, 0.201647], [0,0,0,0], [9E9, 9E9, 9E9, 9E9, 9E9, 9E9]];
	VAR robtarget OpenholeUD_3287 := [[385.33, -25.5, 177.78], [-0.183051, 0.683002, 0.683002, 0.183051], [0,0,0,0], [9E9, 9E9, 9E9, 9E9, 9E9, 9E9]];
	VAR robtarget OpenholeUD_3288 := [[381.33, -25.5, 177.79], [-0.183051, 0.683002, 0.683002, 0.183051], [0,0,0,0], [9E9, 9E9, 9E9, 9E9, 9E9, 9E9]];
	VAR robtarget OpenholeUD_3289 := [[377.33, -25.5, 177.8], [-0.183051, 0.683002, 0.683002, 0.183051], [0,0,0,0], [9E9, 9E9, 9E9, 9E9, 9E9, 9E9]];
	VAR robtarget OpenholeUD_3290 := [[373.33, -25.5, 177.81], [-0.183051, 0.683002, 0.683002, 0.183051], [0,0,0,0], [9E9, 9E9, 9E9, 9E9, 9E9, 9E9]];
	VAR robtarget OpenholeUD_3291 := [[369.33, -25.5, 177.83], [-0.183051, 0.683002, 0.683002, 0.183051], [0,0,0,0], [9E9, 9E9, 9E9, 9E9, 9E9, 9E9]];
	VAR robtarget OpenholeUD_3292 := [[369.33, -25.5, 177.83], [-0.183051, 0.683002, 0.683002, 0.183051], [0,0,0,0], [9E9, 9E9, 9E9, 9E9, 9E9, 9E9]];
	VAR robtarget OpenholeUD_3293 := [[369.34, -24.3, 178.52], [-0.183051, 0.683002, 0.683002, 0.183051], [0,0,0,0], [9E9, 9E9, 9E9, 9E9, 9E9, 9E9]];
	VAR robtarget OpenholeUD_3294 := [[373.34, -24.3, 178.51], [-0.183051, 0.683002, 0.683002, 0.183051], [0,0,0,0], [9E9, 9E9, 9E9, 9E9, 9E9, 9E9]];
	VAR robtarget OpenholeUD_3295 := [[377.34, -24.3, 178.49], [-0.183051, 0.683002, 0.683002, 0.183051], [0,0,0,0], [9E9, 9E9, 9E9, 9E9, 9E9, 9E9]];
	VAR robtarget OpenholeUD_3296 := [[381.34, -24.3, 178.48], [-0.183051, 0.683002, 0.683002, 0.183051], [0,0,0,0], [9E9, 9E9, 9E9, 9E9, 9E9, 9E9]];
	VAR robtarget OpenholeUD_3297 := [[389.34, -24.3, 178.46], [-0.167478, 0.686987, 0.678742, 0.198265], [0,0,0,0], [9E9, 9E9, 9E9, 9E9, 9E9, 9E9]];
	VAR robtarget OpenholeUD_3298 := [[393.33, -24.3, 178.66], [-0.157095, 0.689435, 0.681497, 0.188579], [0,0,0,0], [9E9, 9E9, 9E9, 9E9, 9E9, 9E9]];
	VAR robtarget OpenholeUD_3299 := [[397.33, -24.3, 178.86], [-0.14635, 0.691796, 0.6842, 0.178524], [0,0,0,0], [9E9, 9E9, 9E9, 9E9, 9E9, 9E9]];
	VAR robtarget OpenholeUD_3300 := [[401.32, -24.3, 179.06], [-0.135247, 0.694052, 0.686835, 0.1681], [0,0,0,0], [9E9, 9E9, 9E9, 9E9, 9E9, 9E9]];
	VAR robtarget OpenholeUD_3301 := [[405.32, -24.3, 179.27], [-0.123794, 0.696186, 0.689386, 0.15731], [0,0,0,0], [9E9, 9E9, 9E9, 9E9, 9E9, 9E9]];
	VAR robtarget OpenholeUD_3302 := [[409.31, -24.3, 179.47], [-0.112003, 0.69818, 0.691836, 0.146162], [0,0,0,0], [9E9, 9E9, 9E9, 9E9, 9E9, 9E9]];
	VAR robtarget OpenholeUD_3303 := [[413.31, -24.3, 179.67], [-0.09989, 0.700016, 0.694165, 0.134664], [0,0,0,0], [9E9, 9E9, 9E9, 9E9, 9E9, 9E9]];
	VAR robtarget OpenholeUD_3304 := [[417.3, -24.3, 179.88], [-0.087476, 0.701675, 0.696356, 0.122832], [0,0,0,0], [9E9, 9E9, 9E9, 9E9, 9E9, 9E9]];
	VAR robtarget OpenholeUD_3305 := [[421.3, -24.3, 180.08], [-0.074785, 0.703141, 0.698391, 0.110682], [0,0,0,0], [9E9, 9E9, 9E9, 9E9, 9E9, 9E9]];
	VAR robtarget OpenholeUD_3306 := [[425.29, -24.3, 180.28], [-0.061845, 0.704397, 0.70025, 0.098238], [0,0,0,0], [9E9, 9E9, 9E9, 9E9, 9E9, 9E9]];
	VAR robtarget OpenholeUD_3307 := [[429.29, -24.3, 180.48], [-0.04869, 0.705428, 0.701916, 0.085525], [0,0,0,0], [9E9, 9E9, 9E9, 9E9, 9E9, 9E9]];
	VAR robtarget OpenholeUD_3308 := [[433.28, -24.3, 180.69], [-0.035356, 0.706222, 0.703373, 0.072574], [0,0,0,0], [9E9, 9E9, 9E9, 9E9, 9E9, 9E9]];
	VAR robtarget OpenholeUD_3309 := [[437.28, -24.3, 180.89], [-0.021882, 0.706768, 0.704606, 0.05942], [0,0,0,0], [9E9, 9E9, 9E9, 9E9, 9E9, 9E9]];
	VAR robtarget OpenholeUD_3310 := [[441.27, -24.3, 181.09], [-0.008311, 0.707058, 0.705602, 0.0461], [0,0,0,0], [9E9, 9E9, 9E9, 9E9, 9E9, 9E9]];
	VAR robtarget OpenholeUD_3311 := [[446.05, -24.3, 181.33], [0.007979, 0.707062, 0.706469, 0.030015], [0,0,0,0], [9E9, 9E9, 9E9, 9E9, 9E9, 9E9]];
	VAR robtarget OpenholeUD_3312 := [[446.05, -24.3, 181.33], [0.007979, 0.707062, 0.706469, 0.030015], [0,0,0,0], [9E9, 9E9, 9E9, 9E9, 9E9, 9E9]];
	VAR robtarget OpenholeUD_3313 := [[444.56, -23.1, 181.31], [-0.001167, 0.707106, 0.706428, 0.030973], [0,0,0,0], [9E9, 9E9, 9E9, 9E9, 9E9, 9E9]];
	VAR robtarget OpenholeUD_3314 := [[440.56, -23.1, 181.16], [-0.014782, 0.706952, 0.70571, 0.044421], [0,0,0,0], [9E9, 9E9, 9E9, 9E9, 9E9, 9E9]];
	VAR robtarget OpenholeUD_3315 := [[436.57, -23.1, 181], [-0.028329, 0.706539, 0.704745, 0.057743], [0,0,0,0], [9E9, 9E9, 9E9, 9E9, 9E9, 9E9]];
	VAR robtarget OpenholeUD_3316 := [[432.57, -23.1, 180.84], [-0.041763, 0.705872, 0.703543, 0.070899], [0,0,0,0], [9E9, 9E9, 9E9, 9E9, 9E9, 9E9]];
	VAR robtarget OpenholeUD_3317 := [[428.57, -23.1, 180.69], [-0.055044, 0.704961, 0.702117, 0.083852], [0,0,0,0], [9E9, 9E9, 9E9, 9E9, 9E9, 9E9]];
	VAR robtarget OpenholeUD_3318 := [[424.58, -23.1, 180.53], [-0.068132, 0.703817, 0.700482, 0.096566], [0,0,0,0], [9E9, 9E9, 9E9, 9E9, 9E9, 9E9]];
	VAR robtarget OpenholeUD_3319 := [[420.58, -23.1, 180.37], [-0.080993, 0.702453, 0.698653, 0.109012], [0,0,0,0], [9E9, 9E9, 9E9, 9E9, 9E9, 9E9]];
	VAR robtarget OpenholeUD_3320 := [[416.58, -23.1, 180.22], [-0.093594, 0.700885, 0.696649, 0.121164], [0,0,0,0], [9E9, 9E9, 9E9, 9E9, 9E9, 9E9]];
	VAR robtarget OpenholeUD_3321 := [[412.59, -23.1, 180.06], [-0.105909, 0.69913, 0.694486, 0.132999], [0,0,0,0], [9E9, 9E9, 9E9, 9E9, 9E9, 9E9]];
	VAR robtarget OpenholeUD_3322 := [[408.59, -23.1, 179.9], [-0.117913, 0.697206, 0.692185, 0.1445], [0,0,0,0], [9E9, 9E9, 9E9, 9E9, 9E9, 9E9]];
	VAR robtarget OpenholeUD_3323 := [[404.59, -23.1, 179.75], [-0.129589, 0.695131, 0.689763, 0.155652], [0,0,0,0], [9E9, 9E9, 9E9, 9E9, 9E9, 9E9]];
	VAR robtarget OpenholeUD_3324 := [[400.6, -23.1, 179.59], [-0.140921, 0.692922, 0.687238, 0.166446], [0,0,0,0], [9E9, 9E9, 9E9, 9E9, 9E9, 9E9]];
	VAR robtarget OpenholeUD_3325 := [[396.6, -23.1, 179.43], [-0.151899, 0.690599, 0.684628, 0.176875], [0,0,0,0], [9E9, 9E9, 9E9, 9E9, 9E9, 9E9]];
	VAR robtarget OpenholeUD_3326 := [[389.34, -23.1, 179.15], [-0.170911, 0.686141, 0.679723, 0.194876], [0,0,0,0], [9E9, 9E9, 9E9, 9E9, 9E9, 9E9]];
	VAR robtarget OpenholeUD_3327 := [[385.34, -23.1, 179.16], [-0.183051, 0.683002, 0.683002, 0.183051], [0,0,0,0], [9E9, 9E9, 9E9, 9E9, 9E9, 9E9]];
	VAR robtarget OpenholeUD_3328 := [[381.34, -23.1, 179.17], [-0.183051, 0.683002, 0.683002, 0.183051], [0,0,0,0], [9E9, 9E9, 9E9, 9E9, 9E9, 9E9]];
	VAR robtarget OpenholeUD_3329 := [[377.34, -23.1, 179.19], [-0.183051, 0.683002, 0.683002, 0.183051], [0,0,0,0], [9E9, 9E9, 9E9, 9E9, 9E9, 9E9]];
	VAR robtarget OpenholeUD_3330 := [[373.34, -23.1, 179.2], [-0.183051, 0.683002, 0.683002, 0.183051], [0,0,0,0], [9E9, 9E9, 9E9, 9E9, 9E9, 9E9]];
	VAR robtarget OpenholeUD_3331 := [[369.34, -23.1, 179.21], [-0.183051, 0.683002, 0.683002, 0.183051], [0,0,0,0], [9E9, 9E9, 9E9, 9E9, 9E9, 9E9]];
	VAR robtarget OpenholeUD_3332 := [[369.34, -23.1, 179.21], [-0.183051, 0.683002, 0.683002, 0.183051], [0,0,0,0], [9E9, 9E9, 9E9, 9E9, 9E9, 9E9]];
	VAR robtarget OpenholeUD_3333 := [[369.34, -21.9, 179.9], [-0.183051, 0.683002, 0.683002, 0.183051], [0,0,0,0], [9E9, 9E9, 9E9, 9E9, 9E9, 9E9]];
	VAR robtarget OpenholeUD_3334 := [[373.34, -21.9, 179.89], [-0.183051, 0.683002, 0.683002, 0.183051], [0,0,0,0], [9E9, 9E9, 9E9, 9E9, 9E9, 9E9]];
	VAR robtarget OpenholeUD_3335 := [[377.34, -21.9, 179.88], [-0.183051, 0.683002, 0.683002, 0.183051], [0,0,0,0], [9E9, 9E9, 9E9, 9E9, 9E9, 9E9]];
	VAR robtarget OpenholeUD_3336 := [[381.34, -21.9, 179.87], [-0.183051, 0.683002, 0.683002, 0.183051], [0,0,0,0], [9E9, 9E9, 9E9, 9E9, 9E9, 9E9]];
	VAR robtarget OpenholeUD_3337 := [[385.34, -21.9, 179.85], [-0.183051, 0.683002, 0.683002, 0.183051], [0,0,0,0], [9E9, 9E9, 9E9, 9E9, 9E9, 9E9]];
	VAR robtarget OpenholeUD_3338 := [[389.34, -21.9, 179.84], [-0.174343, 0.685277, 0.680687, 0.19148], [0,0,0,0], [9E9, 9E9, 9E9, 9E9, 9E9, 9E9]];
	VAR robtarget OpenholeUD_3339 := [[393.34, -21.9, 179.95], [-0.164089, 0.687804, 0.683378, 0.181645], [0,0,0,0], [9E9, 9E9, 9E9, 9E9, 9E9, 9E9]];
	VAR robtarget OpenholeUD_3340 := [[397.34, -21.9, 180.06], [-0.15347, 0.690251, 0.686008, 0.171444], [0,0,0,0], [9E9, 9E9, 9E9, 9E9, 9E9, 9E9]];
	VAR robtarget OpenholeUD_3341 := [[401.34, -21.9, 180.17], [-0.142487, 0.692602, 0.688563, 0.160876], [0,0,0,0], [9E9, 9E9, 9E9, 9E9, 9E9, 9E9]];
	VAR robtarget OpenholeUD_3342 := [[405.34, -21.9, 180.28], [-0.13115, 0.694838, 0.691025, 0.149947], [0,0,0,0], [9E9, 9E9, 9E9, 9E9, 9E9, 9E9]];
	VAR robtarget OpenholeUD_3343 := [[409.33, -21.9, 180.39], [-0.119468, 0.696941, 0.693378, 0.138663], [0,0,0,0], [9E9, 9E9, 9E9, 9E9, 9E9, 9E9]];
	VAR robtarget OpenholeUD_3344 := [[413.33, -21.9, 180.51], [-0.107457, 0.698894, 0.695602, 0.127036], [0,0,0,0], [9E9, 9E9, 9E9, 9E9, 9E9, 9E9]];
	VAR robtarget OpenholeUD_3345 := [[417.33, -21.9, 180.62], [-0.095135, 0.700678, 0.697679, 0.115081], [0,0,0,0], [9E9, 9E9, 9E9, 9E9, 9E9, 9E9]];
	VAR robtarget OpenholeUD_3346 := [[421.33, -21.9, 180.73], [-0.082527, 0.702274, 0.699592, 0.102817], [0,0,0,0], [9E9, 9E9, 9E9, 9E9, 9E9, 9E9]];
	VAR robtarget OpenholeUD_3347 := [[425.33, -21.9, 180.84], [-0.069659, 0.703667, 0.701321, 0.090269], [0,0,0,0], [9E9, 9E9, 9E9, 9E9, 9E9, 9E9]];
	VAR robtarget OpenholeUD_3348 := [[429.33, -21.9, 180.95], [-0.056564, 0.704841, 0.702851, 0.077463], [0,0,0,0], [9E9, 9E9, 9E9, 9E9, 9E9, 9E9]];
	VAR robtarget OpenholeUD_3349 := [[433.32, -21.9, 181.06], [-0.043276, 0.705781, 0.704165, 0.064431], [0,0,0,0], [9E9, 9E9, 9E9, 9E9, 9E9, 9E9]];
	VAR robtarget OpenholeUD_3350 := [[437.32, -21.9, 181.17], [-0.029836, 0.706477, 0.70525, 0.051208], [0,0,0,0], [9E9, 9E9, 9E9, 9E9, 9E9, 9E9]];
	VAR robtarget OpenholeUD_3351 := [[443.69, -21.9, 181.34], [-0.008228, 0.707059, 0.706476, 0.029862], [0,0,0,0], [9E9, 9E9, 9E9, 9E9, 9E9, 9E9]];
	VAR robtarget OpenholeUD_3352 := [[443.69, -21.9, 181.34], [-0.008228, 0.707059, 0.706476, 0.029862], [0,0,0,0], [9E9, 9E9, 9E9, 9E9, 9E9, 9E9]];
	VAR robtarget OpenholeUD_3353 := [[443.16, -20.7, 181.4], [-0.014107, 0.706966, 0.706569, 0.02758], [0,0,0,0], [9E9, 9E9, 9E9, 9E9, 9E9, 9E9]];
	VAR robtarget OpenholeUD_3354 := [[439.16, -20.7, 181.34], [-0.027685, 0.706565, 0.705915, 0.04103], [0,0,0,0], [9E9, 9E9, 9E9, 9E9, 9E9, 9E9]];
	VAR robtarget OpenholeUD_3355 := [[435.16, -20.7, 181.27], [-0.041164, 0.705908, 0.705015, 0.054354], [0,0,0,0], [9E9, 9E9, 9E9, 9E9, 9E9, 9E9]];
	VAR robtarget OpenholeUD_3356 := [[431.16, -20.7, 181.21], [-0.054502, 0.705003, 0.703877, 0.067511], [0,0,0,0], [9E9, 9E9, 9E9, 9E9, 9E9, 9E9]];
	VAR robtarget OpenholeUD_3357 := [[427.16, -20.7, 181.14], [-0.067659, 0.703862, 0.702514, 0.080465], [0,0,0,0], [9E9, 9E9, 9E9, 9E9, 9E9, 9E9]];
	VAR robtarget OpenholeUD_3358 := [[423.16, -20.7, 181.08], [-0.080597, 0.702498, 0.70094, 0.093181], [0,0,0,0], [9E9, 9E9, 9E9, 9E9, 9E9, 9E9]];
	VAR robtarget OpenholeUD_3359 := [[419.16, -20.7, 181.02], [-0.093285, 0.700926, 0.699173, 0.105629], [0,0,0,0], [9E9, 9E9, 9E9, 9E9, 9E9, 9E9]];
	VAR robtarget OpenholeUD_3360 := [[415.17, -20.7, 180.95], [-0.105693, 0.699163, 0.697228, 0.117784], [0,0,0,0], [9E9, 9E9, 9E9, 9E9, 9E9, 9E9]];
	VAR robtarget OpenholeUD_3361 := [[411.17, -20.7, 180.89], [-0.117796, 0.697226, 0.695124, 0.129623], [0,0,0,0], [9E9, 9E9, 9E9, 9E9, 9E9, 9E9]];
	VAR robtarget OpenholeUD_3362 := [[407.17, -20.7, 180.82], [-0.129575, 0.695133, 0.69288, 0.141129], [0,0,0,0], [9E9, 9E9, 9E9, 9E9, 9E9, 9E9]];
	VAR robtarget OpenholeUD_3363 := [[403.17, -20.7, 180.76], [-0.141011, 0.692904, 0.690513, 0.152288], [0,0,0,0], [9E9, 9E9, 9E9, 9E9, 9E9, 9E9]];
	VAR robtarget OpenholeUD_3364 := [[399.17, -20.7, 180.69], [-0.152094, 0.690556, 0.688042, 0.16309], [0,0,0,0], [9E9, 9E9, 9E9, 9E9, 9E9, 9E9]];
	VAR robtarget OpenholeUD_3365 := [[395.17, -20.7, 180.63], [-0.162815, 0.688107, 0.685483, 0.173529], [0,0,0,0], [9E9, 9E9, 9E9, 9E9, 9E9, 9E9]];
	VAR robtarget OpenholeUD_3366 := [[389.34, -20.7, 180.53], [-0.177772, 0.684395, 0.681635, 0.188077], [0,0,0,0], [9E9, 9E9, 9E9, 9E9, 9E9, 9E9]];
	VAR robtarget OpenholeUD_3367 := [[385.34, -20.7, 180.55], [-0.183051, 0.683002, 0.683002, 0.183051], [0,0,0,0], [9E9, 9E9, 9E9, 9E9, 9E9, 9E9]];
	VAR robtarget OpenholeUD_3368 := [[381.34, -20.7, 180.56], [-0.183051, 0.683002, 0.683002, 0.183051], [0,0,0,0], [9E9, 9E9, 9E9, 9E9, 9E9, 9E9]];
	VAR robtarget OpenholeUD_3369 := [[377.34, -20.7, 180.57], [-0.183051, 0.683002, 0.683002, 0.183051], [0,0,0,0], [9E9, 9E9, 9E9, 9E9, 9E9, 9E9]];
	VAR robtarget OpenholeUD_3370 := [[373.34, -20.7, 180.59], [-0.183051, 0.683002, 0.683002, 0.183051], [0,0,0,0], [9E9, 9E9, 9E9, 9E9, 9E9, 9E9]];
	VAR robtarget OpenholeUD_3371 := [[369.34, -20.7, 180.6], [-0.183051, 0.683002, 0.683002, 0.183051], [0,0,0,0], [9E9, 9E9, 9E9, 9E9, 9E9, 9E9]];
	VAR robtarget OpenholeUD_3372 := [[369.34, -20.7, 180.6], [-0.183051, 0.683002, 0.683002, 0.183051], [0,0,0,0], [9E9, 9E9, 9E9, 9E9, 9E9, 9E9]];
	VAR robtarget OpenholeUD_3373 := [[369.35, -19.5, 181.29], [-0.183051, 0.683002, 0.683002, 0.183051], [0,0,0,0], [9E9, 9E9, 9E9, 9E9, 9E9, 9E9]];
	VAR robtarget OpenholeUD_3374 := [[373.35, -19.5, 181.28], [-0.183051, 0.683002, 0.683002, 0.183051], [0,0,0,0], [9E9, 9E9, 9E9, 9E9, 9E9, 9E9]];
	VAR robtarget OpenholeUD_3375 := [[377.35, -19.5, 181.27], [-0.183051, 0.683002, 0.683002, 0.183051], [0,0,0,0], [9E9, 9E9, 9E9, 9E9, 9E9, 9E9]];
	VAR robtarget OpenholeUD_3376 := [[381.35, -19.5, 181.25], [-0.183051, 0.683002, 0.683002, 0.183051], [0,0,0,0], [9E9, 9E9, 9E9, 9E9, 9E9, 9E9]];
	VAR robtarget OpenholeUD_3377 := [[385.35, -19.5, 181.24], [-0.183051, 0.683002, 0.683002, 0.183051], [0,0,0,0], [9E9, 9E9, 9E9, 9E9, 9E9, 9E9]];
	VAR robtarget OpenholeUD_3378 := [[389.35, -19.5, 181.23], [-0.181197, 0.683497, 0.682567, 0.184669], [0,0,0,0], [9E9, 9E9, 9E9, 9E9, 9E9, 9E9]];
	VAR robtarget OpenholeUD_3379 := [[393.35, -19.5, 181.25], [-0.171079, 0.686099, 0.685188, 0.174692], [0,0,0,0], [9E9, 9E9, 9E9, 9E9, 9E9, 9E9]];
	VAR robtarget OpenholeUD_3380 := [[397.35, -19.5, 181.26], [-0.160592, 0.688629, 0.687742, 0.164349], [0,0,0,0], [9E9, 9E9, 9E9, 9E9, 9E9, 9E9]];
	VAR robtarget OpenholeUD_3381 := [[401.35, -19.5, 181.28], [-0.149739, 0.69107, 0.690213, 0.153644], [0,0,0,0], [9E9, 9E9, 9E9, 9E9, 9E9, 9E9]];
	VAR robtarget OpenholeUD_3382 := [[405.35, -19.5, 181.3], [-0.138525, 0.693405, 0.692583, 0.142581], [0,0,0,0], [9E9, 9E9, 9E9, 9E9, 9E9, 9E9]];
	VAR robtarget OpenholeUD_3383 := [[409.35, -19.5, 181.32], [-0.126961, 0.695616, 0.694834, 0.131169], [0,0,0,0], [9E9, 9E9, 9E9, 9E9, 9E9, 9E9]];
	VAR robtarget OpenholeUD_3384 := [[413.35, -19.5, 181.34], [-0.11506, 0.697683, 0.69695, 0.11942], [0,0,0,0], [9E9, 9E9, 9E9, 9E9, 9E9, 9E9]];
	VAR robtarget OpenholeUD_3385 := [[417.35, -19.5, 181.36], [-0.10284, 0.699588, 0.69891, 0.107351], [0,0,0,0], [9E9, 9E9, 9E9, 9E9, 9E9, 9E9]];
	VAR robtarget OpenholeUD_3386 := [[421.35, -19.5, 181.37], [-0.090324, 0.701314, 0.700699, 0.094982], [0,0,0,0], [9E9, 9E9, 9E9, 9E9, 9E9, 9E9]];
	VAR robtarget OpenholeUD_3387 := [[425.35, -19.5, 181.39], [-0.077538, 0.702843, 0.702297, 0.082338], [0,0,0,0], [9E9, 9E9, 9E9, 9E9, 9E9, 9E9]];
	VAR robtarget OpenholeUD_3388 := [[429.35, -19.5, 181.41], [-0.064512, 0.704158, 0.703688, 0.069448], [0,0,0,0], [9E9, 9E9, 9E9, 9E9, 9E9, 9E9]];
	VAR robtarget OpenholeUD_3389 := [[433.35, -19.5, 181.43], [-0.051282, 0.705245, 0.704858, 0.056344], [0,0,0,0], [9E9, 9E9, 9E9, 9E9, 9E9, 9E9]];
	VAR robtarget OpenholeUD_3390 := [[437.35, -19.5, 181.45], [-0.037885, 0.706091, 0.705794, 0.043064], [0,0,0,0], [9E9, 9E9, 9E9, 9E9, 9E9, 9E9]];
	VAR robtarget OpenholeUD_3391 := [[442.9, -19.5, 181.47], [-0.019095, 0.706849, 0.706685, 0.024414], [0,0,0,0], [9E9, 9E9, 9E9, 9E9, 9E9, 9E9]];
	VAR robtarget OpenholeUD_3392 := [[442.9, -19.5, 181.47], [-0.019095, 0.706849, 0.706685, 0.024414], [0,0,0,0], [9E9, 9E9, 9E9, 9E9, 9E9, 9E9]];
	VAR robtarget OpenholeUD_3393 := [[442.86, -18.3, 181.55], [-0.023305, 0.706723, 0.70681, 0.020475], [0,0,0,0], [9E9, 9E9, 9E9, 9E9, 9E9, 9E9]];
	VAR robtarget OpenholeUD_3394 := [[438.86, -18.3, 181.57], [-0.036848, 0.706146, 0.706291, 0.033951], [0,0,0,0], [9E9, 9E9, 9E9, 9E9, 9E9, 9E9]];
	VAR robtarget OpenholeUD_3395 := [[434.86, -18.3, 181.6], [-0.050274, 0.705317, 0.705522, 0.047312], [0,0,0,0], [9E9, 9E9, 9E9, 9E9, 9E9, 9E9]];
	VAR robtarget OpenholeUD_3396 := [[430.86, -18.3, 181.63], [-0.063543, 0.704246, 0.704512, 0.060517], [0,0,0,0], [9E9, 9E9, 9E9, 9E9, 9E9, 9E9]];
	VAR robtarget OpenholeUD_3397 := [[426.86, -18.3, 181.66], [-0.076614, 0.702944, 0.703274, 0.073528], [0,0,0,0], [9E9, 9E9, 9E9, 9E9, 9E9, 9E9]];
	VAR robtarget OpenholeUD_3398 := [[422.86, -18.3, 181.69], [-0.089452, 0.701426, 0.701819, 0.086311], [0,0,0,0], [9E9, 9E9, 9E9, 9E9, 9E9, 9E9]];
	VAR robtarget OpenholeUD_3399 := [[418.86, -18.3, 181.71], [-0.102026, 0.699708, 0.700166, 0.098834], [0,0,0,0], [9E9, 9E9, 9E9, 9E9, 9E9, 9E9]];
	VAR robtarget OpenholeUD_3400 := [[414.86, -18.3, 181.74], [-0.114308, 0.697806, 0.698329, 0.111071], [0,0,0,0], [9E9, 9E9, 9E9, 9E9, 9E9, 9E9]];
	VAR robtarget OpenholeUD_3401 := [[410.86, -18.3, 181.77], [-0.126275, 0.69574, 0.696327, 0.123], [0,0,0,0], [9E9, 9E9, 9E9, 9E9, 9E9, 9E9]];
	VAR robtarget OpenholeUD_3402 := [[406.86, -18.3, 181.8], [-0.137908, 0.693528, 0.694178, 0.134601], [0,0,0,0], [9E9, 9E9, 9E9, 9E9, 9E9, 9E9]];
	VAR robtarget OpenholeUD_3403 := [[402.86, -18.3, 181.83], [-0.149192, 0.691189, 0.691899, 0.145861], [0,0,0,0], [9E9, 9E9, 9E9, 9E9, 9E9, 9E9]];
	VAR robtarget OpenholeUD_3404 := [[398.86, -18.3, 181.85], [-0.160116, 0.68874, 0.68951, 0.156768], [0,0,0,0], [9E9, 9E9, 9E9, 9E9, 9E9, 9E9]];
	VAR robtarget OpenholeUD_3405 := [[394.86, -18.3, 181.88], [-0.170674, 0.6862, 0.687027, 0.167315], [0,0,0,0], [9E9, 9E9, 9E9, 9E9, 9E9, 9E9]];
	VAR robtarget OpenholeUD_3406 := [[389.35, -18.3, 181.92], [-0.184618, 0.68258, 0.683481, 0.181256], [0,0,0,0], [9E9, 9E9, 9E9, 9E9, 9E9, 9E9]];
	VAR robtarget OpenholeUD_3407 := [[385.35, -18.3, 181.93], [-0.183051, 0.683002, 0.683002, 0.183051], [0,0,0,0], [9E9, 9E9, 9E9, 9E9, 9E9, 9E9]];
	VAR robtarget OpenholeUD_3408 := [[381.35, -18.3, 181.95], [-0.183051, 0.683002, 0.683002, 0.183051], [0,0,0,0], [9E9, 9E9, 9E9, 9E9, 9E9, 9E9]];
	VAR robtarget OpenholeUD_3409 := [[377.35, -18.3, 181.96], [-0.183051, 0.683002, 0.683002, 0.183051], [0,0,0,0], [9E9, 9E9, 9E9, 9E9, 9E9, 9E9]];
	VAR robtarget OpenholeUD_3410 := [[373.35, -18.3, 181.97], [-0.183051, 0.683002, 0.683002, 0.183051], [0,0,0,0], [9E9, 9E9, 9E9, 9E9, 9E9, 9E9]];
	VAR robtarget OpenholeUD_3411 := [[369.35, -18.3, 181.98], [-0.183051, 0.683002, 0.683002, 0.183051], [0,0,0,0], [9E9, 9E9, 9E9, 9E9, 9E9, 9E9]];
	VAR robtarget OpenholeUD_3412 := [[369.35, -18.3, 181.98], [-0.183051, 0.683002, 0.683002, 0.183051], [0,0,0,0], [9E9, 9E9, 9E9, 9E9, 9E9, 9E9]];
	VAR robtarget OpenholeUD_3413 := [[369.35, -17.1, 182.68], [-0.183051, 0.683002, 0.683002, 0.183051], [0,0,0,0], [9E9, 9E9, 9E9, 9E9, 9E9, 9E9]];
	VAR robtarget OpenholeUD_3414 := [[373.35, -17.1, 182.66], [-0.183051, 0.683002, 0.683002, 0.183051], [0,0,0,0], [9E9, 9E9, 9E9, 9E9, 9E9, 9E9]];
	VAR robtarget OpenholeUD_3415 := [[377.35, -17.1, 182.65], [-0.183051, 0.683002, 0.683002, 0.183051], [0,0,0,0], [9E9, 9E9, 9E9, 9E9, 9E9, 9E9]];
	VAR robtarget OpenholeUD_3416 := [[381.35, -17.1, 182.64], [-0.183051, 0.683002, 0.683002, 0.183051], [0,0,0,0], [9E9, 9E9, 9E9, 9E9, 9E9, 9E9]];
	VAR robtarget OpenholeUD_3417 := [[389.35, -17.1, 182.61], [-0.188035, 0.681647, 0.684378, 0.177839], [0,0,0,0], [9E9, 9E9, 9E9, 9E9, 9E9, 9E9]];
	VAR robtarget OpenholeUD_3418 := [[393.35, -17.1, 182.54], [-0.178058, 0.684321, 0.686927, 0.167724], [0,0,0,0], [9E9, 9E9, 9E9, 9E9, 9E9, 9E9]];
	VAR robtarget OpenholeUD_3419 := [[397.35, -17.1, 182.47], [-0.16771, 0.68693, 0.689401, 0.157248], [0,0,0,0], [9E9, 9E9, 9E9, 9E9, 9E9, 9E9]];
	VAR robtarget OpenholeUD_3420 := [[401.35, -17.1, 182.39], [-0.156992, 0.689459, 0.691783, 0.146411], [0,0,0,0], [9E9, 9E9, 9E9, 9E9, 9E9, 9E9]];
	VAR robtarget OpenholeUD_3421 := [[405.35, -17.1, 182.32], [-0.14591, 0.691889, 0.694057, 0.135222], [0,0,0,0], [9E9, 9E9, 9E9, 9E9, 9E9, 9E9]];
	VAR robtarget OpenholeUD_3422 := [[409.35, -17.1, 182.24], [-0.134472, 0.694203, 0.696205, 0.123689], [0,0,0,0], [9E9, 9E9, 9E9, 9E9, 9E9, 9E9]];
	VAR robtarget OpenholeUD_3423 := [[413.35, -17.1, 182.17], [-0.12269, 0.696382, 0.698208, 0.111827], [0,0,0,0], [9E9, 9E9, 9E9, 9E9, 9E9, 9E9]];
